C05441=1066.388,-25.189,-63.754,172.227,25.150,154.618
C05442=1066.394,-24.939,-63.767,172.229,25.153,154.619
C05443=1066.400,-24.690,-63.780,172.230,25.155,154.619
C05444=1066.407,-24.440,-63.794,172.232,25.157,154.619
C05445=1066.413,-24.190,-63.807,172.233,25.159,154.619
C05446=1066.418,-23.941,-63.821,172.235,25.162,154.620
C05447=1066.424,-23.691,-63.833,172.236,25.164,154.620
C05448=1066.431,-23.442,-63.847,172.238,25.166,154.620
C05449=1066.436,-23.192,-63.860,172.239,25.169,154.620
C05450=1066.442,-22.943,-63.874,172.240,25.171,154.621
C05451=1066.448,-22.694,-63.887,172.242,25.173,154.621
C05452=1066.454,-22.443,-63.901,172.243,25.176,154.621
C05453=1066.460,-22.193,-63.914,172.245,25.178,154.622
C05454=1066.467,-21.944,-63.927,172.246,25.181,154.622
C05455=1066.472,-21.695,-63.941,172.248,25.183,154.622
C05456=1066.478,-21.445,-63.954,172.249,25.185,154.622
C05457=1066.485,-21.196,-63.967,172.251,25.187,154.622
C05458=1066.491,-20.946,-63.982,172.252,25.189,154.623
C05459=1066.496,-20.696,-63.994,172.253,25.192,154.623
C05460=1066.503,-20.447,-64.008,172.255,25.194,154.623
C05461=1066.508,-20.197,-64.021,172.256,25.196,154.624
C05462=1066.514,-19.948,-64.035,172.258,25.199,154.624
C05463=1066.521,-19.698,-64.048,172.259,25.201,154.624
C05464=1066.527,-19.448,-64.062,172.261,25.204,154.624
C05465=1066.533,-19.199,-64.075,172.262,25.206,154.625
C05466=1066.539,-18.950,-64.089,172.263,25.208,154.625
C05467=1066.545,-18.700,-64.103,172.265,25.211,154.625
C05468=1066.551,-18.450,-64.116,172.266,25.213,154.625
C05469=1066.558,-18.172,-64.131,172.268,25.215,154.626
C05470=1066.564,-17.893,-64.146,172.270,25.218,154.626
C05471=1066.571,-17.615,-64.162,172.271,25.221,154.626
C05472=1066.578,-17.338,-64.176,172.273,25.223,154.627
C05473=1066.584,-17.087,-64.190,172.274,25.226,154.627
C05474=1066.591,-16.838,-64.204,172.276,25.228,154.627
C05475=1066.596,-16.589,-64.217,172.277,25.230,154.627
C05476=1066.602,-16.339,-64.231,172.279,25.233,154.628
C05477=1066.609,-16.089,-64.244,172.280,25.235,154.628
C05478=1066.615,-15.840,-64.258,172.282,25.237,154.628
C05479=1066.621,-15.590,-64.272,172.283,25.240,154.628
C05480=1066.627,-15.341,-64.285,172.284,25.242,154.629
C05481=1066.633,-15.091,-64.299,172.286,25.244,154.629
C05482=1066.639,-14.842,-64.312,172.287,25.247,154.629
C05483=1066.645,-14.592,-64.326,172.289,25.249,154.630
C05484=1066.651,-14.342,-64.340,172.290,25.252,154.630
C05485=1066.657,-14.093,-64.354,172.292,25.254,154.630
C05486=1066.663,-13.843,-64.368,172.294,25.257,154.630
C05487=1066.669,-13.594,-64.381,172.295,25.259,154.631
C05488=1066.675,-13.345,-64.395,172.297,25.261,154.631
C05489=1066.681,-13.095,-64.409,172.298,25.264,154.631
C05490=1066.687,-12.845,-64.423,172.300,25.267,154.632
C05491=1066.692,-12.596,-64.437,172.301,25.269,154.632
C05492=1066.699,-12.346,-64.450,172.302,25.271,154.632
C05493=1066.705,-12.096,-64.464,172.304,25.274,154.632
C05494=1066.711,-11.847,-64.478,172.305,25.276,154.633
C05495=1066.717,-11.598,-64.492,172.307,25.278,154.633
C05496=1066.723,-11.348,-64.506,172.308,25.281,154.633
C05497=1066.729,-11.098,-64.520,172.310,25.283,154.633
C05498=1066.734,-10.849,-64.533,172.311,25.286,154.634
C05499=1066.741,-10.599,-64.547,172.312,25.288,154.634
C05500=1066.747,-10.350,-64.562,172.314,25.291,154.634
C05501=1066.752,-10.100,-64.576,172.315,25.293,154.635
C05502=1066.759,-9.850,-64.589,172.317,25.295,154.635
C05503=1066.765,-9.601,-64.603,172.318,25.298,154.635
C05504=1066.771,-9.352,-64.617,172.320,25.300,154.635
C05505=1066.777,-9.102,-64.631,172.321,25.302,154.636
C05506=1066.783,-8.852,-64.645,172.322,25.305,154.636
C05507=1066.789,-8.603,-64.658,172.324,25.308,154.636
C05508=1066.795,-8.353,-64.673,172.325,25.310,154.637
C05509=1066.801,-8.104,-64.687,172.327,25.312,154.637
C05510=1066.807,-7.854,-64.700,172.328,25.315,154.637
C05511=1066.813,-7.604,-64.715,172.330,25.317,154.637
C05512=1066.819,-7.355,-64.729,172.331,25.319,154.638
C05513=1066.825,-7.106,-64.743,172.332,25.322,154.638
C05514=1066.831,-6.856,-64.757,172.334,25.325,154.638
C05515=1066.837,-6.607,-64.771,172.335,25.327,154.639
C05516=1066.844,-6.357,-64.785,172.337,25.329,154.639
C05517=1066.849,-6.107,-64.799,172.338,25.332,154.639
C05518=1066.855,-5.858,-64.813,172.340,25.334,154.640
C05519=1066.862,-5.608,-64.827,172.341,25.336,154.640
C05520=1066.867,-5.359,-64.841,172.342,25.339,154.640
C05521=1066.875,-5.109,-64.855,172.344,25.342,154.640
C05522=1066.880,-4.860,-64.869,172.345,25.344,154.641
C05523=1066.886,-4.611,-64.884,172.347,25.346,154.641
C05524=1066.892,-4.361,-64.898,172.348,25.349,154.641
C05525=1066.898,-4.111,-64.911,172.349,25.351,154.642
C05526=1066.904,-3.862,-64.926,172.351,25.353,154.642
C05527=1066.910,-3.612,-64.940,172.352,25.356,154.642
C05528=1066.917,-3.363,-64.954,172.354,25.359,154.642
C05529=1066.923,-3.113,-64.968,172.355,25.361,154.643
C05530=1066.928,-2.864,-64.982,172.357,25.363,154.643
C05531=1066.934,-2.614,-64.997,172.358,25.366,154.643
C05532=1066.940,-2.364,-65.011,172.359,25.369,154.644
C05533=1066.947,-2.085,-65.027,172.361,25.371,154.644
C05534=1066.953,-1.805,-65.043,172.363,25.374,154.644
C05535=1066.960,-1.525,-65.059,172.364,25.377,154.645
C05536=1066.966,-1.245,-65.075,172.366,25.380,154.645
C05537=1066.973,-0.995,-65.089,172.367,25.382,154.645
C05538=1066.978,-0.746,-65.104,172.369,25.385,154.646
C05539=1066.984,-0.496,-65.118,172.370,25.388,154.646
C05540=1066.990,-0.247,-65.133,172.371,25.390,154.646
C05541=1066.996,0.003,-65.147,172.373,25.392,154.647
C05542=1067.002,0.252,-65.162,172.374,25.395,154.647
C05543=1067.008,0.501,-65.176,172.376,25.398,154.647
C05544=1067.014,0.752,-65.191,172.377,25.400,154.648
C05545=1067.020,1.001,-65.205,172.378,25.402,154.648
C05546=1067.025,1.250,-65.219,172.380,25.405,154.648
C05547=1067.032,1.500,-65.233,172.381,25.408,154.648
C05548=1067.038,1.749,-65.247,172.383,25.410,154.649
C05549=1067.044,1.999,-65.262,172.384,25.413,154.649
C05550=1067.050,2.248,-65.277,172.385,25.415,154.649
C05551=1067.056,2.498,-65.291,172.387,25.417,154.650
C05552=1067.062,2.747,-65.305,172.388,25.420,154.650
C05553=1067.068,2.997,-65.320,172.390,25.423,154.650
C05554=1067.074,3.246,-65.334,172.391,25.425,154.651
C05555=1067.080,3.496,-65.349,172.392,25.428,154.651
C05556=1067.085,3.745,-65.363,172.394,25.430,154.651
C05557=1067.092,3.995,-65.378,172.395,25.433,154.652
C05558=1067.098,4.244,-65.393,172.397,25.436,154.652
C05559=1067.104,4.494,-65.407,172.398,25.438,154.652
C05560=1067.109,4.743,-65.421,172.399,25.440,154.652
C05561=1067.116,4.993,-65.436,172.401,25.443,154.653
C05562=1067.121,5.243,-65.450,172.402,25.446,154.653
C05563=1067.128,5.492,-65.465,172.404,25.448,154.653
C05564=1067.134,5.741,-65.480,172.405,25.451,154.654
C05565=1067.140,5.991,-65.495,172.406,25.453,154.654
C05566=1067.145,6.240,-65.509,172.408,25.455,154.654
C05567=1067.152,6.490,-65.524,172.409,25.458,154.655
C05568=1067.158,6.739,-65.538,172.411,25.461,154.655
C05569=1067.164,6.989,-65.553,172.412,25.463,154.655
C05570=1067.169,7.238,-65.567,172.413,25.466,154.656
C05571=1067.176,7.488,-65.582,172.415,25.468,154.656
C05572=1067.181,7.738,-65.597,172.416,25.471,154.656
C05573=1067.187,7.987,-65.612,172.418,25.474,154.657
C05574=1067.193,8.237,-65.626,172.419,25.476,154.657
C05575=1067.199,8.486,-65.641,172.421,25.478,154.657
C05576=1067.205,8.736,-65.656,172.422,25.481,154.658
C05577=1067.215,9.138,-65.680,172.424,25.485,154.658
C05578=1067.225,9.540,-65.702,172.426,25.489,154.659
C05579=1067.235,9.942,-65.727,172.429,25.493,154.659
C05580=1067.245,10.344,-65.750,172.431,25.497,154.660
C05581=1067.251,10.594,-65.765,172.433,25.499,154.660
C05582=1067.257,10.843,-65.779,172.434,25.502,154.660
C05583=1067.263,11.093,-65.794,172.435,25.505,154.660
C05584=1067.269,11.343,-65.810,172.437,25.507,154.661
C05585=1067.275,11.592,-65.825,172.438,25.510,154.661
C05586=1067.281,11.841,-65.839,172.440,25.512,154.661
C05587=1067.287,12.090,-65.854,172.441,25.515,154.662
C05588=1067.293,12.340,-65.868,172.442,25.518,154.662
C05589=1067.299,12.590,-65.883,172.444,25.520,154.662
C05590=1067.305,12.839,-65.898,172.445,25.522,154.663
C05591=1067.311,13.089,-65.913,172.447,25.525,154.663
C05592=1067.318,13.338,-65.928,172.448,25.527,154.663
C05593=1067.327,13.716,-65.951,172.450,25.531,154.664
C05594=1067.336,14.095,-65.973,172.452,25.535,154.664
C05595=1067.345,14.475,-65.996,172.455,25.539,154.665
C05596=1067.354,14.853,-66.018,172.456,25.543,154.665
C05597=1067.361,15.102,-66.033,172.458,25.546,154.666
C05598=1067.366,15.352,-66.049,172.459,25.548,154.666
C05599=1067.372,15.601,-66.064,172.461,25.551,154.666
C05600=1067.378,15.850,-66.078,172.462,25.553,154.667
C05601=1067.384,16.100,-66.093,172.464,25.556,154.667
C05602=1067.390,16.350,-66.109,172.465,25.558,154.667
C05603=1067.396,16.599,-66.123,172.466,25.561,154.668
C05604=1067.402,16.848,-66.138,172.468,25.564,154.668
C05605=1067.408,17.098,-66.154,172.469,25.566,154.668
C05606=1067.414,17.347,-66.168,172.471,25.569,154.669
C05607=1067.420,17.597,-66.183,172.472,25.572,154.669
C05608=1067.426,17.847,-66.199,172.473,25.574,154.669
C05609=1067.431,18.096,-66.213,172.475,25.577,154.670
C05610=1067.438,18.345,-66.229,172.476,25.579,154.670
C05611=1067.444,18.595,-66.244,172.478,25.582,154.670
C05612=1067.450,18.845,-66.259,172.479,25.584,154.671
C05613=1067.456,19.094,-66.274,172.480,25.587,154.671
C05614=1067.462,19.344,-66.290,172.482,25.590,154.671
C05615=1067.468,19.593,-66.304,172.483,25.592,154.671
C05616=1067.474,19.842,-66.319,172.485,25.595,154.672
C05617=1067.480,20.092,-66.335,172.486,25.597,154.672
C05618=1067.486,20.341,-66.350,172.487,25.600,154.673
C05619=1067.492,20.591,-66.365,172.489,25.602,154.673
C05620=1067.498,20.840,-66.380,172.490,25.605,154.673
C05621=1067.504,21.090,-66.395,172.492,25.608,154.674
C05622=1067.510,21.340,-66.411,172.493,25.611,154.674
C05623=1067.516,21.588,-66.426,172.494,25.613,154.674
C05624=1067.521,21.838,-66.442,172.496,25.616,154.675
C05625=1067.528,22.088,-66.457,172.497,25.618,154.675
C05626=1067.533,22.338,-66.472,172.499,25.621,154.675
C05627=1067.539,22.586,-66.488,172.500,25.623,154.676
C05628=1067.546,22.836,-66.502,172.501,25.626,154.676
C05629=1067.551,23.086,-66.518,172.503,25.629,154.676
C05630=1067.557,23.335,-66.533,172.504,25.631,154.677
C05631=1067.563,23.584,-66.549,172.506,25.634,154.677
C05632=1067.570,23.834,-66.564,172.507,25.637,154.677
C05633=1067.575,24.084,-66.579,172.508,25.639,154.678
C05634=1067.581,24.332,-66.594,172.510,25.642,154.678
C05635=1067.587,24.582,-66.610,172.511,25.644,154.678
C05636=1067.593,24.831,-66.625,172.513,25.647,154.679
C05637=1067.599,25.081,-66.641,172.514,25.649,154.679
C05638=1067.606,25.331,-66.656,172.515,25.652,154.679
C05639=1067.611,25.580,-66.671,172.517,25.655,154.680
C05640=1067.617,25.829,-66.686,172.518,25.658,154.680
C05641=1067.623,26.079,-66.703,172.520,25.660,154.680
C05642=1067.629,26.328,-66.718,172.521,25.663,154.681
C05643=1067.635,26.578,-66.733,172.522,25.665,154.681
C05644=1067.641,26.827,-66.748,172.524,25.668,154.681
C05645=1067.647,27.077,-66.764,172.525,25.670,154.682
C05646=1067.653,27.326,-66.780,172.527,25.673,154.682
C05647=1067.659,27.576,-66.795,172.528,25.676,154.682
C05648=1067.665,27.825,-66.810,172.529,25.678,154.683
C05649=1067.671,28.074,-66.826,172.531,25.681,154.683
C05650=1067.676,28.324,-66.842,172.532,25.684,154.683
C05651=1067.683,28.573,-66.857,172.533,25.687,154.684
C05652=1067.689,28.823,-66.873,172.535,25.689,154.684
C05653=1067.695,29.072,-66.888,172.536,25.692,154.684
C05654=1067.701,29.322,-66.904,172.538,25.694,154.685
C05655=1067.706,29.571,-66.920,172.539,25.697,154.685
C05656=1067.713,29.820,-66.935,172.540,25.700,154.685
C05657=1067.720,30.103,-66.952,172.542,25.703,154.686
C05658=1067.726,30.387,-66.970,172.543,25.706,154.686
C05659=1067.733,30.670,-66.988,172.544,25.709,154.687
C05660=1067.740,30.954,-67.006,172.547,25.712,154.687
C05661=1067.745,31.202,-67.022,172.548,25.714,154.687
C05662=1067.751,31.452,-67.037,172.550,25.717,154.688
C05663=1067.757,31.702,-67.054,172.551,25.720,154.688
C05664=1067.763,31.951,-67.068,172.552,25.722,154.688
C05665=1067.769,32.201,-67.085,172.554,25.725,154.689
C05666=1067.775,32.451,-67.100,172.554,25.727,154.689
C05667=1067.782,32.700,-67.116,172.556,25.730,154.689
C05668=1067.787,32.948,-67.132,172.557,25.733,154.690
C05669=1067.793,33.198,-67.147,172.558,25.735,154.690
C05670=1067.799,33.448,-67.164,172.560,25.738,154.691
C05671=1067.805,33.697,-67.179,172.561,25.740,154.691
C05672=1067.811,33.947,-67.195,172.563,25.743,154.691
C05673=1067.817,34.196,-67.211,172.564,25.746,154.692
C05674=1067.823,34.446,-67.226,172.565,25.748,154.692
C05675=1067.829,34.695,-67.242,172.567,25.751,154.692
C05676=1067.835,34.945,-67.258,172.568,25.754,154.693
C05677=1067.840,35.194,-67.274,172.570,25.757,154.693
C05678=1067.847,35.443,-67.289,172.571,25.759,154.693
C05679=1067.853,35.693,-67.305,172.572,25.762,154.694
C05680=1067.859,35.942,-67.321,172.574,25.765,154.694
C05681=1067.864,36.191,-67.337,172.575,25.767,154.694
C05682=1067.871,36.441,-67.352,172.577,25.770,154.695
C05683=1067.877,36.690,-67.369,172.578,25.772,154.695
C05684=1067.883,36.940,-67.385,172.579,25.775,154.695
C05685=1067.888,37.190,-67.400,172.581,25.777,154.696
C05686=1067.895,37.439,-67.416,172.582,25.780,154.696
C05687=1067.901,37.688,-67.432,172.584,25.783,154.696
C05688=1067.907,37.937,-67.449,172.585,25.785,154.697
C05689=1067.913,38.187,-67.464,172.586,25.788,154.697
C05690=1067.919,38.437,-67.480,172.588,25.791,154.697
C05691=1067.924,38.685,-67.496,172.589,25.794,154.698
C05692=1067.930,38.935,-67.513,172.591,25.796,154.698
C05693=1067.936,39.185,-67.528,172.592,25.799,154.698
C05694=1067.941,39.434,-67.544,172.593,25.802,154.699
C05695=1067.947,39.683,-67.561,172.595,25.805,154.699
C05696=1067.953,39.933,-67.577,172.596,25.807,154.700
C05697=1067.960,40.182,-67.593,172.598,25.810,154.700
C05698=1067.966,40.432,-67.608,172.599,25.813,154.700
C05699=1067.972,40.681,-67.624,172.600,25.815,154.701
C05700=1067.978,40.930,-67.641,172.602,25.818,154.701
C05701=1067.984,41.180,-67.657,172.603,25.821,154.701
C05702=1067.990,41.429,-67.673,172.605,25.823,154.702
C05703=1067.995,41.678,-67.689,172.606,25.826,154.702
C05704=1068.001,41.928,-67.705,172.607,25.829,154.702
C05705=1068.007,42.178,-67.721,172.609,25.831,154.703
C05706=1068.013,42.427,-67.737,172.610,25.834,154.703
C05707=1068.019,42.676,-67.754,172.611,25.837,154.704
C05708=1068.025,42.926,-67.770,172.613,25.839,154.704
C05709=1068.031,43.175,-67.786,172.614,25.842,154.704
C05710=1068.037,43.424,-67.802,172.616,25.844,154.705
C05711=1068.043,43.674,-67.819,172.617,25.847,154.705
C05712=1068.049,43.923,-67.835,172.618,25.850,154.705
C05713=1068.054,44.173,-67.850,172.620,25.853,154.706
C05714=1068.060,44.422,-67.867,172.621,25.855,154.706
C05715=1068.066,44.672,-67.884,172.623,25.858,154.706
C05716=1068.071,44.921,-67.900,172.624,25.861,154.707
C05717=1068.077,45.170,-67.916,172.625,25.864,154.707
C05718=1068.083,45.419,-67.932,172.627,25.866,154.707
C05719=1068.089,45.669,-67.948,172.628,25.869,154.708
C05720=1068.095,45.918,-67.964,172.630,25.872,154.708
C05721=1068.101,46.202,-67.984,172.631,25.875,154.709
C05722=1068.107,46.485,-68.002,172.633,25.878,154.709
C05723=1068.114,46.768,-68.020,172.634,25.881,154.710
C05724=1068.121,47.051,-68.040,172.636,25.884,154.710
C05725=1068.127,47.301,-68.056,172.637,25.887,154.710
C05726=1068.133,47.550,-68.072,172.639,25.890,154.711
C05727=1068.139,47.799,-68.089,172.640,25.892,154.711
C05728=1068.144,48.049,-68.105,172.641,25.895,154.711
C05729=1068.150,48.298,-68.122,172.643,25.898,154.712
C05730=1068.156,48.548,-68.138,172.644,25.900,154.712
C05731=1068.162,48.797,-68.154,172.646,25.903,154.712
C05732=1068.167,49.047,-68.171,172.647,25.906,154.713
C05733=1068.173,49.296,-68.187,172.648,25.909,154.713
C05734=1068.179,49.545,-68.204,172.650,25.911,154.714
C05735=1068.185,49.794,-68.221,172.651,25.914,154.714
C05736=1068.191,50.043,-68.237,172.653,25.917,154.714
C05737=1068.197,50.293,-68.254,172.654,25.919,154.715
C05738=1068.203,50.543,-68.270,172.655,25.922,154.715
C05739=1068.209,50.792,-68.286,172.657,25.925,154.715
C05740=1068.215,51.042,-68.303,172.658,25.927,154.716
C05741=1068.220,51.292,-68.320,172.660,25.930,154.716
C05742=1068.227,51.540,-68.337,172.661,25.933,154.716
C05743=1068.233,51.790,-68.353,172.662,25.936,154.717
C05744=1068.238,52.039,-68.369,172.664,25.938,154.717
C05745=1068.244,52.289,-68.386,172.665,25.941,154.718
C05746=1068.250,52.538,-68.402,172.667,25.944,154.718
C05747=1068.256,52.787,-68.418,172.668,25.946,154.718
C05748=1068.262,53.036,-68.435,172.669,25.949,154.719
C05749=1068.267,53.286,-68.452,172.671,25.952,154.719
C05750=1068.274,53.536,-68.469,172.672,25.955,154.719
C05751=1068.280,53.785,-68.485,172.674,25.957,154.720
C05752=1068.286,54.034,-68.502,172.675,25.960,154.720
C05753=1068.291,54.284,-68.519,172.676,25.963,154.720
C05754=1068.297,54.533,-68.535,172.678,25.965,154.721
C05755=1068.303,54.782,-68.552,172.679,25.968,154.721
C05756=1068.308,55.031,-68.569,172.681,25.971,154.722
C05757=1068.315,55.281,-68.586,172.682,25.973,154.722
C05758=1068.321,55.531,-68.602,172.683,25.976,154.722
C05759=1068.327,55.779,-68.619,172.685,25.979,154.723
C05760=1068.332,56.029,-68.636,172.686,25.982,154.723
C05761=1068.338,56.278,-68.652,172.688,25.984,154.723
C05762=1068.345,56.527,-68.669,172.689,25.987,154.724
C05763=1068.350,56.777,-68.686,172.690,25.990,154.724
C05764=1068.356,57.027,-68.702,172.692,25.992,154.724
C05765=1068.363,57.276,-68.719,172.693,25.995,154.725
C05766=1068.369,57.525,-68.736,172.695,25.998,154.725
C05767=1068.374,57.775,-68.753,172.696,26.000,154.726
C05768=1068.381,58.024,-68.770,172.697,26.003,154.726
C05769=1068.387,58.273,-68.786,172.699,26.006,154.726
C05770=1068.392,58.523,-68.803,172.700,26.008,154.727
C05771=1068.398,58.772,-68.820,172.703,26.011,154.727
C05772=1068.405,59.022,-68.837,172.704,26.014,154.727
C05773=1068.410,59.271,-68.854,172.705,26.017,154.728
C05774=1068.416,59.520,-68.870,172.707,26.019,154.728
C05775=1068.422,59.770,-68.887,172.708,26.022,154.728
C05776=1068.428,60.019,-68.905,172.710,26.025,154.729
C05777=1068.434,60.269,-68.921,172.711,26.027,154.729
C05778=1068.440,60.517,-68.938,172.713,26.030,154.729
C05779=1068.446,60.767,-68.955,172.714,26.033,154.730
C05780=1068.452,61.016,-68.972,172.715,26.035,154.730
C05781=1068.458,61.266,-68.988,172.717,26.038,154.730
C05782=1068.464,61.515,-69.006,172.718,26.041,154.731
C05783=1068.470,61.764,-69.022,172.720,26.043,154.731
C05784=1068.477,62.014,-69.039,172.721,26.046,154.732
C05785=1068.483,62.296,-69.058,172.722,26.049,154.732
C05786=1068.490,62.580,-69.078,172.724,26.052,154.732
C05787=1068.496,62.862,-69.097,172.726,26.055,154.733
C05788=1068.504,63.145,-69.116,172.727,26.058,154.733
C05789=1068.509,63.395,-69.134,172.729,26.061,154.734
C05790=1068.516,63.645,-69.150,172.730,26.063,154.734
C05791=1068.521,63.894,-69.168,172.732,26.066,154.734
C05792=1068.527,64.143,-69.184,172.733,26.069,154.735
C05793=1068.534,64.392,-69.202,172.735,26.071,154.735
C05794=1068.539,64.642,-69.218,172.736,26.074,154.735
C05795=1068.546,64.891,-69.235,172.737,26.077,154.736
C05796=1068.551,65.140,-69.253,172.739,26.079,154.736
C05797=1068.557,65.390,-69.270,172.740,26.082,154.736
C05798=1068.563,65.639,-69.287,172.742,26.085,154.737
C05799=1068.568,65.889,-69.304,172.743,26.088,154.737
C05800=1068.575,66.138,-69.321,172.744,26.090,154.737
C05801=1068.581,66.387,-69.339,172.746,26.093,154.738
C05802=1068.586,66.637,-69.356,172.747,26.096,154.738
C05803=1068.592,66.885,-69.373,172.749,26.098,154.739
C05804=1068.598,67.135,-69.391,172.750,26.101,154.739
C05805=1068.604,67.385,-69.407,172.751,26.104,154.739
C05806=1068.610,67.634,-69.424,172.753,26.107,154.740
C05807=1068.616,67.883,-69.442,172.754,26.109,154.740
C05808=1068.622,68.133,-69.459,172.756,26.112,154.740
C05809=1068.628,68.382,-69.476,172.757,26.115,154.741
C05810=1068.634,68.631,-69.494,172.759,26.117,154.741
C05811=1068.640,68.880,-69.511,172.760,26.120,154.741
C05812=1068.645,69.130,-69.528,172.761,26.123,154.742
C05813=1068.651,69.380,-69.546,172.763,26.125,154.742
C05814=1068.657,69.628,-69.563,172.764,26.128,154.743
C05815=1068.663,69.877,-69.580,172.767,26.131,154.743
C05816=1068.669,70.128,-69.598,172.768,26.134,154.743
C05817=1068.675,70.376,-69.615,172.769,26.137,154.744
C05818=1068.681,70.625,-69.632,172.771,26.139,154.744
C05819=1068.687,70.875,-69.650,172.772,26.142,154.744
C05820=1068.692,71.124,-69.668,172.774,26.145,154.745
C05821=1068.698,71.374,-69.684,172.775,26.147,154.745
C05822=1068.704,71.623,-69.702,172.776,26.150,154.745
C05823=1068.710,71.872,-69.719,172.778,26.153,154.746
C05824=1068.715,72.121,-69.737,172.779,26.155,154.746
C05825=1068.722,72.371,-69.754,172.781,26.158,154.747
C05826=1068.728,72.620,-69.772,172.782,26.161,154.747
C05827=1068.734,72.870,-69.789,172.783,26.163,154.747
C05828=1068.739,73.119,-69.807,172.785,26.166,154.748
C05829=1068.745,73.368,-69.824,172.786,26.169,154.748
C05830=1068.751,73.618,-69.842,172.788,26.171,154.748
C05831=1068.757,73.867,-69.859,172.789,26.174,154.749
C05832=1068.762,74.116,-69.877,172.791,26.177,154.749
C05833=1068.769,74.366,-69.895,172.792,26.179,154.750
C05834=1068.774,74.615,-69.912,172.793,26.182,154.750
C05835=1068.780,74.864,-69.930,172.795,26.185,154.750
C05836=1068.786,75.113,-69.947,172.796,26.188,154.751
C05837=1068.792,75.362,-69.965,172.798,26.190,154.751
C05838=1068.798,75.612,-69.983,172.799,26.193,154.751
C05839=1068.803,75.862,-70.000,172.800,26.196,154.752
C05840=1068.809,76.111,-70.017,172.802,26.198,154.752
C05841=1068.815,76.360,-70.035,172.803,26.201,154.753
C05842=1068.822,76.610,-70.052,172.805,26.204,154.753
C05843=1068.827,76.859,-70.070,172.806,26.207,154.753
C05844=1068.833,77.109,-70.088,172.808,26.209,154.754
C05845=1068.839,77.358,-70.105,172.810,26.212,154.754
C05846=1068.845,77.607,-70.123,172.811,26.215,154.754
C05847=1068.851,77.856,-70.141,172.813,26.217,154.755
C05848=1068.856,78.105,-70.158,172.814,26.220,154.755
C05849=1068.863,78.388,-70.179,172.816,26.223,154.755
C05850=1068.870,78.671,-70.199,172.817,26.227,154.756
C05851=1068.876,78.954,-70.219,172.819,26.230,154.756
C05852=1068.883,79.237,-70.239,172.821,26.233,154.757
C05853=1068.889,79.486,-70.256,172.822,26.235,154.757
C05854=1068.895,79.735,-70.275,172.823,26.238,154.758
C05855=1068.901,79.984,-70.293,172.825,26.241,154.758
C05856=1068.907,80.234,-70.311,172.826,26.243,154.758
C05857=1068.912,80.483,-70.328,172.828,26.246,154.759
C05858=1068.919,80.732,-70.346,172.829,26.249,154.759
C05859=1068.923,80.982,-70.364,172.830,26.252,154.759
C05860=1068.929,81.232,-70.382,172.832,26.255,154.760
C05861=1068.935,81.481,-70.400,172.833,26.257,154.760
C05862=1068.941,81.729,-70.418,172.835,26.260,154.761
C05863=1068.947,81.979,-70.436,172.836,26.263,154.761
C05864=1068.952,82.228,-70.454,172.838,26.266,154.761
C05865=1068.959,82.478,-70.472,172.840,26.268,154.762
C05866=1068.964,82.727,-70.489,172.841,26.271,154.762
C05867=1068.970,82.976,-70.508,172.843,26.274,154.762
C05868=1068.976,83.225,-70.525,172.844,26.277,154.763
C05869=1068.982,83.474,-70.543,172.846,26.279,154.763
C05870=1068.988,83.724,-70.561,172.847,26.282,154.763
C05871=1068.993,83.974,-70.579,172.848,26.285,154.764
C05872=1068.999,84.222,-70.598,172.850,26.288,154.764
C05873=1069.005,84.472,-70.616,172.851,26.290,154.765
C05874=1069.010,84.721,-70.633,172.853,26.293,154.765
C05875=1069.017,84.971,-70.651,172.854,26.295,154.765
C05876=1069.023,85.220,-70.670,172.856,26.298,154.766
C05877=1069.029,85.469,-70.687,172.857,26.301,154.766
C05878=1069.035,85.718,-70.705,172.858,26.303,154.766
C05879=1069.040,85.967,-70.723,172.860,26.306,154.767
C05880=1069.046,86.217,-70.742,172.861,26.309,154.767
C05881=1069.051,86.466,-70.760,172.863,26.311,154.768
C05882=1069.058,86.715,-70.778,172.865,26.315,154.768
C05883=1069.063,86.964,-70.796,172.866,26.317,154.768
C05884=1069.069,87.214,-70.814,172.868,26.320,154.769
C05885=1069.076,87.463,-70.832,172.869,26.323,154.769
C05886=1069.081,87.712,-70.850,172.871,26.325,154.769
C05887=1069.088,87.962,-70.868,172.872,26.328,154.770
C05888=1069.093,88.210,-70.887,172.874,26.331,154.770
C05889=1069.099,88.460,-70.905,172.875,26.333,154.770
C05890=1069.105,88.710,-70.923,172.876,26.336,154.771
C05891=1069.111,88.958,-70.941,172.878,26.338,154.771
C05892=1069.117,89.208,-70.959,172.879,26.341,154.772
C05893=1069.123,89.457,-70.977,172.881,26.344,154.772
C05894=1069.129,89.706,-70.995,172.882,26.346,154.772
C05895=1069.134,89.956,-71.014,172.884,26.349,154.773
C05896=1069.140,90.205,-71.032,172.886,26.352,154.773
C05897=1069.146,90.454,-71.050,172.888,26.355,154.773
C05898=1069.152,90.704,-71.068,172.889,26.358,154.774
C05899=1069.158,90.953,-71.086,172.890,26.360,154.774
C05900=1069.164,91.202,-71.105,172.892,26.363,154.774
C05901=1069.169,91.451,-71.123,172.893,26.365,154.775
C05902=1069.175,91.701,-71.142,172.895,26.368,154.775
C05903=1069.181,91.950,-71.160,172.896,26.371,154.776
C05904=1069.187,92.199,-71.178,172.898,26.374,154.776
C05905=1069.192,92.449,-71.197,172.899,26.377,154.776
C05906=1069.198,92.697,-71.215,172.900,26.379,154.777
C05907=1069.204,92.947,-71.233,172.902,26.382,154.777
C05908=1069.210,93.196,-71.252,172.903,26.385,154.777
C05909=1069.215,93.445,-71.270,172.905,26.388,154.778
C05910=1069.221,93.695,-71.289,172.907,26.390,154.778
C05911=1069.227,93.943,-71.307,172.908,26.393,154.779
C05912=1069.233,94.193,-71.325,172.910,26.396,154.779
C05913=1069.240,94.476,-71.347,172.911,26.399,154.779
C05914=1069.246,94.759,-71.367,172.913,26.402,154.780
C05915=1069.253,95.041,-71.389,172.915,26.405,154.780
C05916=1069.259,95.325,-71.409,172.916,26.408,154.781
C05917=1069.266,95.574,-71.428,172.918,26.411,154.781
C05918=1069.271,95.823,-71.447,172.919,26.413,154.781
C05919=1069.277,96.072,-71.465,172.921,26.416,154.782
C05920=1069.282,96.322,-71.484,172.923,26.419,154.782
C05921=1069.288,96.570,-71.502,172.924,26.422,154.782
C05922=1069.294,96.820,-71.521,172.926,26.424,154.783
C05923=1069.300,97.069,-71.539,172.927,26.427,154.783
C05924=1069.306,97.318,-71.558,172.929,26.430,154.784
C05925=1069.311,97.568,-71.576,172.930,26.433,154.784
C05926=1069.318,97.817,-71.595,172.932,26.435,154.784
C05927=1069.323,98.066,-71.614,172.933,26.438,154.785
C05928=1069.329,98.315,-71.632,172.935,26.441,154.785
C05929=1069.335,98.565,-71.651,172.936,26.443,154.785
C05930=1069.341,98.814,-71.670,172.937,26.446,154.786
C05931=1069.346,99.063,-71.689,172.940,26.449,154.786
C05932=1069.352,99.312,-71.706,172.941,26.451,154.786
C05933=1069.359,99.562,-71.725,172.943,26.454,154.787
C05934=1069.364,99.811,-71.744,172.944,26.457,154.787
C05935=1069.370,100.059,-71.763,172.946,26.460,154.788
C05936=1069.376,100.309,-71.782,172.947,26.462,154.788
C05937=1069.382,100.559,-71.800,172.948,26.465,154.788
C05938=1069.388,100.808,-71.819,172.950,26.468,154.789
C05939=1069.394,101.057,-71.838,172.951,26.470,154.789
C05940=1069.399,101.306,-71.857,172.954,26.473,154.789
C05941=1069.405,101.555,-71.876,172.955,26.476,154.790
C05942=1069.411,101.805,-71.894,172.957,26.479,154.790
C05943=1069.416,102.054,-71.913,172.958,26.481,154.790
C05944=1069.422,102.303,-71.932,172.960,26.484,154.791
C05945=1069.428,102.552,-71.951,172.961,26.487,154.791
C05946=1069.434,102.802,-71.970,172.962,26.489,154.792
C05947=1069.439,103.051,-71.989,172.964,26.492,154.792
C05948=1069.445,103.300,-72.007,172.965,26.495,154.792
C05949=1069.451,103.549,-72.027,172.967,26.497,154.793
C05950=1069.457,103.799,-72.046,172.969,26.500,154.793
C05951=1069.462,104.048,-72.063,172.970,26.503,154.794
C05952=1069.468,104.297,-72.083,172.972,26.506,154.794
C05953=1069.474,104.546,-72.102,172.973,26.508,154.794
C05954=1069.480,104.796,-72.120,172.975,26.511,154.795
C05955=1069.486,105.045,-72.140,172.976,26.514,154.795
C05956=1069.491,105.294,-72.159,172.978,26.516,154.795
C05957=1069.497,105.543,-72.177,172.979,26.519,154.796
C05958=1069.503,105.792,-72.196,172.982,26.522,154.796
C05959=1069.509,106.042,-72.216,172.983,26.525,154.797
C05960=1069.514,106.291,-72.235,172.984,26.527,154.797
C05961=1069.520,106.540,-72.253,172.986,26.530,154.797
C05962=1069.526,106.789,-72.272,172.987,26.533,154.798
C05963=1069.532,107.038,-72.292,172.989,26.535,154.798
C05964=1069.538,107.288,-72.310,172.990,26.538,154.798
C05965=1069.544,107.537,-72.330,172.992,26.541,154.799
C05966=1069.549,107.786,-72.348,172.994,26.544,154.799
C05967=1069.554,108.035,-72.368,172.996,26.546,154.799
C05968=1069.561,108.284,-72.386,172.997,26.549,154.800
C05969=1069.567,108.534,-72.406,172.998,26.552,154.800
C05970=1069.573,108.782,-72.426,173.000,26.554,154.800
C05971=1069.578,109.032,-72.445,173.001,26.557,154.801
C05972=1069.585,109.281,-72.463,173.003,26.560,154.801
C05973=1069.590,109.530,-72.483,173.004,26.562,154.802
C05974=1069.595,109.779,-72.502,173.007,26.565,154.802
C05975=1069.601,110.029,-72.521,173.008,26.568,154.802
C05976=1069.608,110.278,-72.539,173.009,26.571,154.803
C05977=1069.614,110.561,-72.561,173.011,26.574,154.803
C05978=1069.621,110.844,-72.583,173.013,26.577,154.803
C05979=1069.628,111.126,-72.605,173.015,26.580,154.804
C05980=1069.634,111.409,-72.627,173.017,26.583,154.804
C05981=1069.639,111.658,-72.646,173.018,26.586,154.805
C05982=1069.645,111.908,-72.666,173.020,26.588,154.805
C05983=1069.652,112.157,-72.684,173.021,26.591,154.805
C05984=1069.657,112.406,-72.704,173.023,26.594,154.806
C05985=1069.663,112.655,-72.724,173.024,26.596,154.806
C05986=1069.669,112.905,-72.743,173.026,26.599,154.807
C05987=1069.675,113.154,-72.762,173.028,26.602,154.807
C05988=1069.680,113.404,-72.781,173.030,26.605,154.807
C05989=1069.686,113.652,-72.801,173.031,26.607,154.808
C05990=1069.691,113.901,-72.820,173.033,26.610,154.808
C05991=1069.697,114.150,-72.839,173.034,26.612,154.808
C05992=1069.703,114.399,-72.859,173.035,26.615,154.809
C05993=1069.709,114.649,-72.879,173.038,26.618,154.809
C05994=1069.714,114.898,-72.898,173.039,26.621,154.810
C05995=1069.720,115.148,-72.917,173.041,26.623,154.810
C05996=1069.726,115.396,-72.937,173.042,26.626,154.810
C05997=1069.732,115.646,-72.956,173.044,26.629,154.811
C05998=1069.737,115.895,-72.976,173.045,26.632,154.811
C05999=1069.743,116.143,-72.995,173.046,26.635,154.811
C06000=1069.749,116.393,-73.014,173.049,26.637,154.812
C06001=1069.755,116.642,-73.034,173.050,26.640,154.812
C06002=1069.760,116.891,-73.054,173.052,26.643,154.812
C06003=1069.765,117.141,-73.073,173.053,26.646,154.813
C06004=1069.771,117.390,-73.093,173.055,26.649,154.813
C06005=1069.777,117.639,-73.113,173.056,26.651,154.814
C06006=1069.783,117.888,-73.133,173.059,26.654,154.814
C06007=1069.789,118.137,-73.152,173.060,26.657,154.814
C06008=1069.794,118.387,-73.171,173.061,26.660,154.815
C06009=1069.800,118.636,-73.191,173.063,26.662,154.815
C06010=1069.805,118.885,-73.211,173.064,26.665,154.815
C06011=1069.811,119.134,-73.231,173.066,26.667,154.816
C06012=1069.817,119.384,-73.250,173.068,26.671,154.816
C06013=1069.822,119.632,-73.270,173.070,26.673,154.817
C06014=1069.828,119.881,-73.289,173.071,26.676,154.817
C06015=1069.834,120.130,-73.309,173.073,26.678,154.817
C06016=1069.839,120.380,-73.329,173.074,26.681,154.818
C06017=1069.845,120.628,-73.349,173.075,26.684,154.818
C06018=1069.851,120.878,-73.368,173.078,26.687,154.818
C06019=1069.857,121.127,-73.388,173.079,26.689,154.819
C06020=1069.862,121.376,-73.407,173.081,26.692,154.819
C06021=1069.868,121.625,-73.427,173.082,26.695,154.820
C06022=1069.873,121.875,-73.447,173.084,26.697,154.820
C06023=1069.879,122.124,-73.467,173.086,26.700,154.820
C06024=1069.885,122.372,-73.487,173.088,26.703,154.821
C06025=1069.891,122.622,-73.506,173.089,26.705,154.821
C06026=1069.897,122.871,-73.526,173.090,26.708,154.821
C06027=1069.903,123.121,-73.546,173.092,26.711,154.822
C06028=1069.908,123.370,-73.566,173.094,26.714,154.822
C06029=1069.914,123.619,-73.586,173.096,26.716,154.822
C06030=1069.920,123.868,-73.605,173.097,26.719,154.823
C06031=1069.926,124.117,-73.625,173.099,26.722,154.823
C06032=1069.932,124.366,-73.645,173.100,26.724,154.824
C06033=1069.937,124.615,-73.665,173.103,26.727,154.824
C06034=1069.943,124.864,-73.685,173.104,26.730,154.824
C06035=1069.949,125.114,-73.704,173.105,26.733,154.825
C06036=1069.955,125.362,-73.724,173.107,26.735,154.825
C06037=1069.961,125.611,-73.744,173.108,26.738,154.825
C06038=1069.966,125.861,-73.764,173.111,26.741,154.826
C06039=1069.972,126.110,-73.784,173.112,26.743,154.826
C06040=1069.978,126.359,-73.804,173.114,26.746,154.826
C06041=1069.985,126.642,-73.827,173.115,26.749,154.827
C06042=1069.991,126.925,-73.849,173.118,26.752,154.827
C06043=1069.997,127.208,-73.872,173.119,26.755,154.828
C06044=1070.004,127.491,-73.895,173.121,26.759,154.828
C06045=1070.010,127.739,-73.915,173.123,26.761,154.828
C06046=1070.016,127.989,-73.934,173.124,26.764,154.829
C06047=1070.021,128.238,-73.955,173.127,26.767,154.829
C06048=1070.027,128.487,-73.975,173.128,26.769,154.829
C06049=1070.034,128.736,-73.995,173.130,26.772,154.830
C06050=1070.040,128.985,-74.015,173.131,26.774,154.830
C06051=1070.045,129.235,-74.035,173.134,26.777,154.831
C06052=1070.051,129.484,-74.055,173.135,26.780,154.831
C06053=1070.057,129.733,-74.075,173.137,26.782,154.831
C06054=1070.063,129.981,-74.095,173.138,26.785,154.832
C06055=1070.068,130.231,-74.116,173.139,26.788,154.832
C06056=1070.074,130.480,-74.136,173.142,26.790,154.832
C06057=1070.080,130.729,-74.155,173.143,26.793,154.833
C06058=1070.086,130.978,-74.175,173.145,26.795,154.833
C06059=1070.091,131.227,-74.195,173.146,26.798,154.833
C06060=1070.098,131.477,-74.216,173.149,26.801,154.834
C06061=1070.104,131.726,-74.236,173.150,26.804,154.834
C06062=1070.109,131.975,-74.256,173.152,26.806,154.834
C06063=1070.115,132.224,-74.276,173.153,26.809,154.835
C06064=1070.121,132.473,-74.297,173.156,26.812,154.835
C06065=1070.127,132.722,-74.317,173.157,26.815,154.836
C06066=1070.132,132.971,-74.338,173.159,26.817,154.836
C06067=1070.138,133.220,-74.358,173.160,26.820,154.836
C06068=1070.144,133.469,-74.378,173.163,26.823,154.837
C06069=1070.150,133.718,-74.398,173.164,26.825,154.837
C06070=1070.155,133.967,-74.419,173.165,26.828,154.837
C06071=1070.161,134.217,-74.439,173.167,26.831,154.838
C06072=1070.167,134.466,-74.460,173.168,26.833,154.838
C06073=1070.173,134.715,-74.480,173.171,26.836,154.838
C06074=1070.178,134.964,-74.500,173.172,26.839,154.839
C06075=1070.184,135.213,-74.520,173.174,26.841,154.839
C06076=1070.190,135.463,-74.541,173.175,26.844,154.840
C06077=1070.196,135.711,-74.561,173.178,26.847,154.840
C06078=1070.201,135.960,-74.581,173.179,26.850,154.840
C06079=1070.206,136.210,-74.602,173.181,26.852,154.841
C06080=1070.213,136.459,-74.622,173.183,26.855,154.841
C06081=1070.218,136.708,-74.643,173.184,26.858,154.841
C06082=1070.224,136.957,-74.663,173.186,26.860,154.842
C06083=1070.229,137.206,-74.683,173.187,26.863,154.842
C06084=1070.236,137.455,-74.704,173.190,26.866,154.843
C06085=1070.242,137.704,-74.725,173.191,26.869,154.843
C06086=1070.247,137.953,-74.746,173.193,26.871,154.843
C06087=1070.253,138.202,-74.766,173.194,26.874,154.844
C06088=1070.259,138.452,-74.786,173.197,26.877,154.844
C06089=1070.265,138.701,-74.806,173.198,26.880,154.844
C06090=1070.270,138.949,-74.828,173.200,26.882,154.845
C06091=1070.275,139.198,-74.848,173.201,26.885,154.845
C06092=1070.282,139.448,-74.869,173.204,26.888,154.845
C06093=1070.287,139.697,-74.889,173.205,26.890,154.846
C06094=1070.293,139.946,-74.910,173.207,26.893,154.846
C06095=1070.299,140.195,-74.931,173.209,26.896,154.846
C06096=1070.305,140.444,-74.951,173.210,26.899,154.847
C06097=1070.310,140.693,-74.972,173.212,26.901,154.847
C06098=1070.315,140.942,-74.992,173.213,26.904,154.848
C06099=1070.322,141.191,-75.013,173.216,26.907,154.848
C06100=1070.327,141.440,-75.034,173.217,26.909,154.848
C06101=1070.333,141.690,-75.054,173.219,26.912,154.849
C06102=1070.338,141.939,-75.075,173.221,26.915,154.849
C06103=1070.345,142.188,-75.096,173.223,26.918,154.849
C06104=1070.350,142.437,-75.117,173.224,26.920,154.850
C06105=1070.357,142.719,-75.141,173.227,26.923,154.850
C06106=1070.363,143.002,-75.164,173.228,26.926,154.851
C06107=1070.369,143.285,-75.187,173.230,26.930,154.851
C06108=1070.376,143.567,-75.211,173.233,26.933,154.851
C06109=1070.381,143.817,-75.232,173.234,26.936,154.852
C06110=1070.387,144.066,-75.253,173.236,26.938,154.852
C06111=1070.393,144.315,-75.274,173.237,26.941,154.853
C06112=1070.399,144.564,-75.294,173.240,26.944,154.853
C06113=1070.405,144.813,-75.315,173.241,26.946,154.853
C06114=1070.410,145.062,-75.336,173.243,26.949,154.854
C06115=1070.416,145.311,-75.358,173.245,26.952,154.854
C06116=1070.422,145.560,-75.378,173.247,26.954,154.854
C06117=1070.427,145.809,-75.399,173.248,26.957,154.855
C06118=1070.434,146.058,-75.420,173.250,26.960,154.855
C06119=1070.439,146.307,-75.441,173.252,26.963,154.855
C06120=1070.445,146.556,-75.462,173.253,26.965,154.856
C06121=1070.450,146.806,-75.482,173.256,26.968,154.856
C06122=1070.456,147.054,-75.504,173.257,26.971,154.857
C06123=1070.462,147.304,-75.525,173.259,26.973,154.857
C06124=1070.468,147.552,-75.545,173.261,26.976,154.857
C06125=1070.473,147.801,-75.566,173.263,26.979,154.858
C06126=1070.480,148.051,-75.588,173.264,26.981,154.858
C06127=1070.485,148.299,-75.609,173.266,26.984,154.858
C06128=1070.491,148.549,-75.630,173.268,26.987,154.859
C06129=1070.497,148.798,-75.651,173.270,26.990,154.859
C06130=1070.502,149.047,-75.672,173.271,26.992,154.859
C06131=1070.508,149.296,-75.693,173.273,26.995,154.860
C06132=1070.513,149.545,-75.714,173.275,26.998,154.860
C06133=1070.519,149.794,-75.735,173.277,27.000,154.860
C06134=1070.525,150.043,-75.757,173.279,27.003,154.861
C06135=1070.531,150.293,-75.778,173.280,27.006,154.861
C06136=1070.536,150.541,-75.799,173.282,27.009,154.862
C06137=1070.542,150.790,-75.819,173.284,27.011,154.862
C06138=1070.548,151.039,-75.841,173.286,27.014,154.862
C06139=1070.553,151.288,-75.862,173.288,27.017,154.863
C06140=1070.559,151.538,-75.883,173.290,27.020,154.863
C06141=1070.565,151.786,-75.904,173.291,27.022,154.863
C06142=1070.571,152.035,-75.926,173.294,27.025,154.864
C06143=1070.576,152.285,-75.947,173.295,27.028,154.864
C06144=1070.582,152.533,-75.968,173.297,27.031,154.865
C06145=1070.588,152.782,-75.990,173.299,27.033,154.865
C06146=1070.593,153.031,-76.011,173.301,27.036,154.865
C06147=1070.599,153.281,-76.032,173.302,27.039,154.866
C06148=1070.604,153.529,-76.054,173.304,27.042,154.866
C06149=1070.610,153.779,-76.075,173.306,27.044,154.866
C06150=1070.616,154.027,-76.097,173.307,27.047,154.867
C06151=1070.622,154.277,-76.117,173.310,27.050,154.867
C06152=1070.627,154.525,-76.139,173.311,27.052,154.867
C06153=1070.633,154.775,-76.160,173.313,27.055,154.868
C06154=1070.639,155.023,-76.182,173.315,27.058,154.868
C06155=1070.645,155.272,-76.203,173.317,27.060,154.868
C06156=1070.650,155.521,-76.224,173.319,27.064,154.869
C06157=1070.656,155.771,-76.246,173.321,27.066,154.869
C06158=1070.661,156.019,-76.267,173.322,27.069,154.870
C06159=1070.668,156.269,-76.289,173.325,27.072,154.870
C06160=1070.673,156.517,-76.310,173.326,27.074,154.870
C06161=1070.679,156.766,-76.332,173.328,27.077,154.871
C06162=1070.684,157.015,-76.354,173.330,27.080,154.871
C06163=1070.690,157.265,-76.375,173.332,27.082,154.871
C06164=1070.696,157.514,-76.396,173.334,27.086,154.872
C06165=1070.702,157.763,-76.418,173.335,27.088,154.872
C06166=1070.707,158.012,-76.440,173.337,27.091,154.873
C06167=1070.713,158.261,-76.461,173.339,27.094,154.873
C06168=1070.719,158.510,-76.483,173.341,27.096,154.873
C06169=1070.725,158.793,-76.507,173.343,27.099,154.874
C06170=1070.731,159.074,-76.532,173.346,27.103,154.874
C06171=1070.738,159.357,-76.556,173.347,27.106,154.875
C06172=1070.744,159.639,-76.580,173.350,27.109,154.875
C06173=1070.750,159.889,-76.602,173.351,27.112,154.875
C06174=1070.756,160.137,-76.623,173.353,27.114,154.876
C06175=1070.761,160.387,-76.646,173.355,27.117,154.876
C06176=1070.768,160.636,-76.667,173.357,27.120,154.876
C06177=1070.773,160.884,-76.688,173.359,27.123,154.877
C06178=1070.779,161.134,-76.710,173.360,27.125,154.877
C06179=1070.784,161.382,-76.732,173.363,27.128,154.877
C06180=1070.790,161.632,-76.754,173.364,27.131,154.878
C06181=1070.795,161.880,-76.775,173.367,27.134,154.878
C06182=1070.802,162.129,-76.798,173.368,27.137,154.879
C06183=1070.807,162.379,-76.820,173.371,27.140,154.879
C06184=1070.812,162.627,-76.842,173.372,27.143,154.879
C06185=1070.818,162.877,-76.864,173.374,27.145,154.880
C06186=1070.823,163.125,-76.885,173.376,27.148,154.880
C06187=1070.829,163.375,-76.907,173.378,27.151,154.881
C06188=1070.834,163.623,-76.929,173.380,27.154,154.881
C06189=1070.840,163.872,-76.951,173.381,27.156,154.881
C06190=1070.845,164.121,-76.973,173.383,27.159,154.882
C06191=1070.850,164.370,-76.995,173.385,27.162,154.882
C06192=1070.857,164.620,-77.017,173.387,27.165,154.883
C06193=1070.861,164.868,-77.039,173.389,27.168,154.883
C06194=1070.868,165.117,-77.061,173.391,27.170,154.883
C06195=1070.873,165.366,-77.083,173.393,27.173,154.884
C06196=1070.878,165.615,-77.105,173.395,27.176,154.884
C06197=1070.884,165.864,-77.127,173.396,27.179,154.884
C06198=1070.889,166.113,-77.150,173.399,27.182,154.885
C06199=1070.896,166.362,-77.171,173.400,27.185,154.885
C06200=1070.900,166.611,-77.193,173.402,27.188,154.886
C06201=1070.906,166.860,-77.215,173.404,27.190,154.886
C06202=1070.912,167.109,-77.238,173.406,27.193,154.886
C06203=1070.917,167.358,-77.259,173.408,27.196,154.887
C06204=1070.923,167.607,-77.282,173.410,27.199,154.887
C06205=1070.929,167.856,-77.304,173.412,27.202,154.887
C06206=1070.934,168.105,-77.326,173.413,27.204,154.888
C06207=1070.940,168.354,-77.348,173.416,27.207,154.888
C06208=1070.946,168.603,-77.370,173.417,27.210,154.889
C06209=1070.951,168.851,-77.392,173.420,27.213,154.889
C06210=1070.957,169.101,-77.414,173.421,27.215,154.889
C06211=1070.963,169.350,-77.437,173.424,27.219,154.890
C06212=1070.967,169.598,-77.459,173.425,27.221,154.890
C06213=1070.974,169.847,-77.481,173.428,27.224,154.891
C06214=1070.979,170.096,-77.503,173.429,27.227,154.891
C06215=1070.984,170.345,-77.525,173.432,27.230,154.891
C06216=1070.991,170.594,-77.548,173.433,27.232,154.892
C06217=1070.996,170.843,-77.570,173.435,27.235,154.892
C06218=1071.002,171.092,-77.593,173.437,27.238,154.892
C06219=1071.007,171.341,-77.614,173.439,27.241,154.893
C06220=1071.013,171.590,-77.637,173.441,27.243,154.893
C06221=1071.018,171.839,-77.659,173.443,27.246,154.893
C06222=1071.025,172.088,-77.682,173.445,27.249,154.894
C06223=1071.030,172.337,-77.703,173.446,27.252,154.894
C06224=1071.035,172.585,-77.726,173.449,27.255,154.895
C06225=1071.042,172.835,-77.748,173.450,27.257,154.895
C06226=1071.047,173.084,-77.771,173.453,27.260,154.895
C06227=1071.052,173.332,-77.793,173.454,27.263,154.896
C06228=1071.058,173.581,-77.816,173.457,27.266,154.896
C06229=1071.064,173.831,-77.837,173.458,27.269,154.897
C06230=1071.070,174.079,-77.860,173.461,27.271,154.897
C06231=1071.075,174.328,-77.883,173.462,27.274,154.897
C06232=1071.081,174.577,-77.905,173.465,27.277,154.898
C06233=1071.087,174.859,-77.930,173.467,27.280,154.898
C06234=1071.094,175.141,-77.955,173.469,27.284,154.898
C06235=1071.100,175.423,-77.982,173.472,27.287,154.899
C06236=1071.107,175.705,-78.007,173.473,27.290,154.899
C06237=1071.113,175.954,-78.030,173.476,27.293,154.900
C06238=1071.119,176.203,-78.051,173.477,27.295,154.900
C06239=1071.124,176.452,-78.074,173.480,27.298,154.900
C06240=1071.130,176.701,-78.097,173.481,27.301,154.901
C06241=1071.136,176.951,-78.119,173.484,27.304,154.901
C06242=1071.141,177.198,-78.141,173.485,27.306,154.902
C06243=1071.147,177.447,-78.164,173.488,27.309,154.902
C06244=1071.153,177.697,-78.187,173.490,27.312,154.902
C06245=1071.158,177.946,-78.210,173.492,27.315,154.903
C06246=1071.164,178.195,-78.232,173.494,27.318,154.903
C06247=1071.171,178.443,-78.255,173.495,27.321,154.903
C06248=1071.176,178.693,-78.277,173.498,27.323,154.904
C06249=1071.182,178.942,-78.300,173.499,27.326,154.904
C06250=1071.187,179.191,-78.323,173.502,27.329,154.904
C06251=1071.194,179.439,-78.345,173.503,27.332,154.905
C06252=1071.199,179.688,-78.367,173.506,27.335,154.905
C06253=1071.204,179.937,-78.390,173.507,27.337,154.905
C06254=1071.210,180.186,-78.413,173.510,27.340,154.906
C06255=1071.216,180.435,-78.436,173.512,27.343,154.906
C06256=1071.222,180.683,-78.458,173.514,27.346,154.907
C06257=1071.228,180.932,-78.481,173.516,27.348,154.907
C06258=1071.234,181.181,-78.504,173.518,27.351,154.907
C06259=1071.239,181.431,-78.526,173.520,27.354,154.908
C06260=1071.245,181.679,-78.549,173.522,27.357,154.908
C06261=1071.251,181.928,-78.572,173.524,27.359,154.908
C06262=1071.257,182.177,-78.595,173.527,27.362,154.909
C06263=1071.263,182.426,-78.618,173.528,27.365,154.909
C06264=1071.269,182.675,-78.641,173.531,27.368,154.910
C06265=1071.274,182.924,-78.664,173.532,27.370,154.910
C06266=1071.281,183.172,-78.686,173.535,27.373,154.910
C06267=1071.287,183.421,-78.709,173.536,27.376,154.911
C06268=1071.292,183.670,-78.732,173.539,27.379,154.911
C06269=1071.298,183.919,-78.755,173.541,27.381,154.911
C06270=1071.304,184.168,-78.778,173.543,27.384,154.912
C06271=1071.310,184.417,-78.801,173.545,27.387,154.912
C06272=1071.315,184.666,-78.824,173.547,27.389,154.912
C06273=1071.321,184.914,-78.847,173.549,27.392,154.913
C06274=1071.327,185.163,-78.869,173.552,27.396,154.913
C06275=1071.332,185.412,-78.892,173.553,27.398,154.914
C06276=1071.338,185.661,-78.915,173.555,27.401,154.914
C06277=1071.343,185.910,-78.939,173.557,27.404,154.914
C06278=1071.349,186.159,-78.962,173.559,27.407,154.915
C06279=1071.355,186.408,-78.985,173.561,27.410,154.915
C06280=1071.360,186.657,-79.008,173.563,27.413,154.916
C06281=1071.365,186.906,-79.031,173.566,27.416,154.916
C06282=1071.371,187.155,-79.055,173.567,27.419,154.916
C06283=1071.377,187.403,-79.078,173.570,27.422,154.917
C06284=1071.382,187.653,-79.101,173.571,27.424,154.917
C06285=1071.388,187.902,-79.124,173.574,27.427,154.918
C06286=1071.394,188.150,-79.147,173.576,27.430,154.918
C06287=1071.399,188.399,-79.170,173.578,27.433,154.918
C06288=1071.405,188.648,-79.195,173.580,27.436,154.919
C06289=1071.410,188.897,-79.217,173.583,27.439,154.919
C06290=1071.416,189.146,-79.240,173.584,27.442,154.920
C06291=1071.421,189.395,-79.264,173.586,27.445,154.920
C06292=1071.427,189.643,-79.288,173.588,27.448,154.920
C06293=1071.433,189.892,-79.311,173.590,27.451,154.921
C06294=1071.439,190.141,-79.334,173.593,27.454,154.921
C06295=1071.444,190.390,-79.357,173.594,27.457,154.921
C06296=1071.450,190.638,-79.381,173.597,27.460,154.922
C06297=1071.456,190.920,-79.407,173.599,27.463,154.922
C06298=1071.462,191.202,-79.433,173.602,27.466,154.923
C06299=1071.468,191.484,-79.460,173.604,27.470,154.923
C06300=1071.475,191.766,-79.486,173.606,27.473,154.924
C06301=1071.481,192.014,-79.510,173.609,27.476,154.924
C06302=1071.486,192.263,-79.533,173.610,27.479,154.924
C06303=1071.492,192.512,-79.556,173.613,27.482,154.925
C06304=1071.498,192.760,-79.580,173.614,27.484,154.925
C06305=1071.503,193.009,-79.604,173.617,27.487,154.926
C06306=1071.509,193.258,-79.627,173.619,27.490,154.926
C06307=1071.514,193.508,-79.651,173.621,27.493,154.926
C06308=1071.520,193.757,-79.674,173.623,27.496,154.927
C06309=1071.526,194.005,-79.698,173.626,27.499,154.927
C06310=1071.531,194.254,-79.721,173.627,27.502,154.928
C06311=1071.537,194.502,-79.745,173.630,27.505,154.928
C06312=1071.543,194.751,-79.768,173.632,27.508,154.928
C06313=1071.548,195.000,-79.792,173.633,27.511,154.929
C06314=1071.554,195.249,-79.815,173.636,27.514,154.929
C06315=1071.560,195.498,-79.839,173.638,27.517,154.930
C06316=1071.565,195.747,-79.863,173.640,27.519,154.930
C06317=1071.571,195.995,-79.886,173.642,27.522,154.930
C06318=1071.576,196.244,-79.910,173.645,27.525,154.931
C06319=1071.582,196.493,-79.934,173.647,27.528,154.931
C06320=1071.589,196.742,-79.957,173.649,27.531,154.932
C06321=1071.594,196.991,-79.981,173.651,27.534,154.932
C06322=1071.600,197.240,-80.004,173.654,27.537,154.932
C06323=1071.605,197.488,-80.028,173.655,27.540,154.933
C06324=1071.611,197.737,-80.052,173.658,27.543,154.933
C06325=1071.617,197.986,-80.076,173.660,27.546,154.934
C06326=1071.623,198.235,-80.100,173.662,27.549,154.934
C06327=1071.629,198.484,-80.122,173.664,27.552,154.934
C06328=1071.634,198.732,-80.147,173.667,27.555,154.935
C06329=1071.640,198.981,-80.171,173.669,27.558,154.935
C06330=1071.645,199.230,-80.194,173.670,27.560,154.935
C06331=1071.651,199.479,-80.218,173.673,27.563,154.936
C06332=1071.657,199.727,-80.242,173.675,27.566,154.936
C06333=1071.663,199.977,-80.266,173.677,27.569,154.937
C06334=1071.669,200.225,-80.289,173.679,27.572,154.937
C06335=1071.674,200.474,-80.313,173.682,27.575,154.937
C06336=1071.681,200.722,-80.337,173.684,27.578,154.938
C06337=1071.686,200.972,-80.361,173.686,27.581,154.938
C06338=1071.692,201.220,-80.385,173.688,27.584,154.939
C06339=1071.697,201.469,-80.409,173.691,27.587,154.939
C06340=1071.704,201.718,-80.433,173.693,27.590,154.939
C06341=1071.709,201.967,-80.456,173.695,27.593,154.940
C06342=1071.715,202.215,-80.480,173.697,27.596,154.940
C06343=1071.721,202.465,-80.505,173.700,27.599,154.941
C06344=1071.727,202.713,-80.528,173.701,27.601,154.941
C06345=1071.732,202.961,-80.553,173.704,27.604,154.941
C06346=1071.738,203.210,-80.577,173.706,27.607,154.942
C06347=1071.743,203.460,-80.601,173.708,27.610,154.942
C06348=1071.749,203.708,-80.625,173.710,27.613,154.943
C06349=1071.755,203.957,-80.649,173.712,27.616,154.943
C06350=1071.760,204.206,-80.673,173.715,27.620,154.943
C06351=1071.766,204.455,-80.698,173.717,27.623,154.944
C06352=1071.772,204.703,-80.721,173.719,27.626,154.944
C06353=1071.777,204.951,-80.746,173.721,27.629,154.945
C06354=1071.783,205.201,-80.770,173.724,27.632,154.945
C06355=1071.788,205.449,-80.794,173.726,27.635,154.945
C06356=1071.794,205.698,-80.818,173.729,27.638,154.946
C06357=1071.800,205.947,-80.843,173.730,27.641,154.946
C06358=1071.806,206.196,-80.867,173.733,27.644,154.947
C06359=1071.811,206.444,-80.891,173.735,27.647,154.947
C06360=1071.817,206.693,-80.915,173.737,27.650,154.948
C06361=1071.841,207.735,-81.017,173.869,27.718,154.949
C06362=1071.851,208.156,-81.059,173.872,27.725,154.950
C06363=1071.861,208.576,-81.102,173.876,27.731,154.951
C06364=1071.871,208.997,-81.144,173.879,27.738,154.953
C06365=1071.880,209.418,-81.186,173.882,27.745,154.954
C06366=1071.886,209.667,-81.211,173.885,27.748,154.954
C06367=1071.892,209.916,-81.236,173.887,27.752,154.955
C06368=1071.898,210.164,-81.261,173.889,27.756,154.955
C06369=1071.904,210.412,-81.286,173.891,27.760,154.956
C06370=1071.910,210.661,-81.311,173.893,27.764,154.957
C06371=1071.916,210.910,-81.336,173.895,27.768,154.957
C06372=1071.921,211.159,-81.362,173.897,27.772,154.958
C06373=1071.927,211.407,-81.387,173.899,27.776,154.959
C06374=1071.933,211.657,-81.412,173.901,27.780,154.959
C06375=1071.939,211.905,-81.436,173.903,27.784,154.960
C06376=1071.945,212.153,-81.462,173.906,27.788,154.960
C06377=1071.951,212.402,-81.487,173.907,27.792,154.961
C06378=1071.956,212.651,-81.513,173.909,27.796,154.962
C06379=1071.962,212.900,-81.537,173.912,27.800,154.962
C06380=1071.968,213.148,-81.563,173.914,27.804,154.963
C06381=1071.974,213.397,-81.588,173.915,27.807,154.964
C06382=1071.979,213.645,-81.614,173.918,27.811,154.964
C06383=1071.985,213.894,-81.639,173.920,27.815,154.965
C06384=1071.991,214.142,-81.664,173.922,27.819,154.965
C06385=1071.997,214.391,-81.690,173.924,27.823,154.966
C06386=1072.002,214.640,-81.714,173.926,27.827,154.967
C06387=1072.008,214.889,-81.740,173.928,27.831,154.967
C06388=1072.014,215.138,-81.766,173.931,27.835,154.968
C06389=1072.020,215.386,-81.791,173.933,27.839,154.969
C06390=1072.026,215.634,-81.816,173.934,27.843,154.969
C06391=1072.031,215.883,-81.842,173.937,27.847,154.970
C06392=1072.037,216.132,-81.867,173.939,27.851,154.970
C06393=1072.044,216.381,-81.893,173.941,27.855,154.971
C06394=1072.049,216.630,-81.919,173.943,27.859,154.972
C06395=1072.055,216.878,-81.944,173.945,27.863,154.972
C06396=1072.061,217.126,-81.969,173.947,27.867,154.973
C06397=1072.066,217.375,-81.995,173.950,27.870,154.974
C06398=1072.073,217.624,-82.020,173.952,27.874,154.974
C06399=1072.078,217.873,-82.046,173.953,27.878,154.975
C06400=1072.084,218.121,-82.071,173.956,27.882,154.975
C06401=1072.090,218.370,-82.096,173.958,27.886,154.976
C06402=1072.095,218.619,-82.122,173.960,27.890,154.977
C06403=1072.101,218.867,-82.148,173.963,27.894,154.977
C06404=1072.108,219.115,-82.174,173.964,27.898,154.978
C06405=1072.113,219.364,-82.200,173.966,27.902,154.979
C06406=1072.120,219.613,-82.225,173.969,27.906,154.979
C06407=1072.125,219.862,-82.251,173.971,27.910,154.980
C06408=1072.131,220.110,-82.276,173.973,27.913,154.980
C06409=1072.136,220.359,-82.302,173.975,27.917,154.981
C06410=1072.142,220.607,-82.327,173.977,27.921,154.982
C06411=1072.149,220.856,-82.353,173.979,27.925,154.982
C06412=1072.154,221.104,-82.379,173.982,27.929,154.983
C06413=1072.161,221.353,-82.405,173.984,27.933,154.983
C06414=1072.165,221.566,-82.427,173.985,27.936,154.984
C06415=1072.171,221.778,-82.449,173.988,27.940,154.985
C06416=1072.175,221.991,-82.471,173.989,27.943,154.985
C06417=1072.180,222.204,-82.494,173.991,27.946,154.986
C06418=1072.186,222.416,-82.515,173.993,27.950,154.986
C06419=1072.190,222.628,-82.537,173.995,27.953,154.987
C06420=1072.195,222.841,-82.560,173.997,27.956,154.987
C06421=1072.200,223.054,-82.582,173.999,27.960,154.988
C06422=1072.206,223.303,-82.608,174.001,27.964,154.988
C06423=1072.212,223.551,-82.633,174.003,27.968,154.989
C06424=1072.218,223.800,-82.660,174.005,27.971,154.990
C06425=1072.223,224.049,-82.686,174.007,27.975,154.990
C06426=1072.229,224.297,-82.711,174.009,27.979,154.991
C06427=1072.235,224.546,-82.738,174.012,27.983,154.991
C06428=1072.241,224.795,-82.763,174.014,27.987,154.992
C06429=1072.247,225.043,-82.790,174.016,27.991,154.993
C06430=1072.253,225.292,-82.815,174.019,27.995,154.993
C06431=1072.258,225.541,-82.841,174.020,27.999,154.994
C06432=1072.264,225.788,-82.867,174.022,28.002,154.995
C06433=1072.269,226.037,-82.893,174.025,28.006,154.995
C06434=1072.275,226.285,-82.920,174.027,28.010,154.996
C06435=1072.281,226.534,-82.945,174.029,28.015,154.996
C06436=1072.287,226.782,-82.972,174.032,28.019,154.997
C06437=1072.293,227.031,-82.998,174.033,28.022,154.998
C06438=1072.299,227.280,-83.025,174.035,28.026,154.998
C06439=1072.305,227.529,-83.050,174.038,28.030,154.999
C06440=1072.311,227.777,-83.077,174.040,28.034,155.000
C06441=1072.316,228.026,-83.103,174.043,28.037,155.000
C06442=1072.323,228.274,-83.129,174.045,28.041,155.001
C06443=1072.328,228.523,-83.155,174.047,28.046,155.001
C06444=1072.334,228.772,-83.181,174.050,28.050,155.002
C06445=1072.340,229.020,-83.208,174.051,28.053,155.003
C06446=1072.346,229.269,-83.233,174.053,28.057,155.003
C06447=1072.352,229.517,-83.260,174.056,28.061,155.004
C06448=1072.358,229.765,-83.286,174.058,28.065,155.004
C06449=1072.363,230.014,-83.312,174.060,28.068,155.005
C06450=1072.370,230.263,-83.338,174.063,28.072,155.006
C06451=1072.376,230.511,-83.365,174.065,28.076,155.006
C06452=1072.381,230.760,-83.391,174.067,28.080,155.007
C06453=1072.387,231.008,-83.418,174.069,28.084,155.008
C06454=1072.393,231.257,-83.445,174.071,28.088,155.008
C06455=1072.399,231.506,-83.471,174.074,28.092,155.009
C06456=1072.404,231.755,-83.497,174.076,28.096,155.009
C06457=1072.410,232.003,-83.524,174.078,28.100,155.010
C06458=1072.416,232.251,-83.551,174.081,28.104,155.011
C06459=1072.421,232.500,-83.576,174.083,28.108,155.011
C06460=1072.427,232.749,-83.603,174.085,28.111,155.012
C06461=1072.433,232.997,-83.630,174.088,28.115,155.012
C06462=1072.439,233.245,-83.656,174.089,28.119,155.013
C06463=1072.446,233.494,-83.683,174.091,28.123,155.014
C06464=1072.452,233.743,-83.709,174.094,28.127,155.014
C06465=1072.457,233.991,-83.735,174.096,28.131,155.015
C06466=1072.462,234.240,-83.763,174.099,28.135,155.016
C06467=1072.468,234.489,-83.789,174.101,28.139,155.016
C06468=1072.474,234.737,-83.816,174.103,28.143,155.017
C06469=1072.479,234.985,-83.843,174.106,28.147,155.017
C06470=1072.489,235.402,-83.887,174.110,28.153,155.018
C06471=1072.499,235.819,-83.932,174.114,28.160,155.020
C06472=1072.509,236.236,-83.977,174.116,28.166,155.021
C06473=1072.519,236.653,-84.022,174.120,28.173,155.022
C06474=1072.525,236.902,-84.049,174.123,28.176,155.022
C06475=1072.531,237.150,-84.075,174.125,28.180,155.023
C06476=1072.537,237.398,-84.102,174.128,28.184,155.023
C06477=1072.542,237.647,-84.129,174.130,28.188,155.024
C06478=1072.548,237.896,-84.156,174.132,28.192,155.025
C06479=1072.554,238.145,-84.183,174.135,28.196,155.025
C06480=1072.560,238.393,-84.210,174.137,28.200,155.026
C06481=1072.565,238.641,-84.236,174.139,28.204,155.027
C06482=1072.572,238.890,-84.263,174.142,28.208,155.027
C06483=1072.578,239.139,-84.290,174.144,28.211,155.028
C06484=1072.584,239.386,-84.317,174.147,28.215,155.028
C06485=1072.589,239.635,-84.344,174.149,28.219,155.029
C06486=1072.595,239.884,-84.372,174.151,28.223,155.030
C06487=1072.601,240.132,-84.398,174.154,28.227,155.030
C06488=1072.607,240.381,-84.425,174.155,28.231,155.031
C06489=1072.613,240.629,-84.452,174.157,28.235,155.031
C06490=1072.619,240.878,-84.479,174.160,28.239,155.032
C06491=1072.624,241.126,-84.507,174.162,28.243,155.033
C06492=1072.630,241.375,-84.533,174.165,28.246,155.033
C06493=1072.636,241.624,-84.560,174.167,28.250,155.034
C06494=1072.642,241.871,-84.588,174.169,28.254,155.035
C06495=1072.648,242.120,-84.614,174.172,28.258,155.035
C06496=1072.654,242.369,-84.642,174.174,28.262,155.036
C06497=1072.660,242.617,-84.669,174.176,28.266,155.036
C06498=1072.666,242.865,-84.696,174.179,28.270,155.037
C06499=1072.671,243.114,-84.723,174.181,28.274,155.038
C06500=1072.677,243.362,-84.751,174.184,28.277,155.038
C06501=1072.683,243.611,-84.777,174.186,28.281,155.039
C06502=1072.688,243.859,-84.805,174.188,28.285,155.039
C06503=1072.695,244.108,-84.832,174.191,28.289,155.040
C06504=1072.700,244.357,-84.860,174.193,28.293,155.041
C06505=1072.706,244.604,-84.887,174.195,28.297,155.041
C06506=1072.712,244.853,-84.914,174.198,28.301,155.042
C06507=1072.718,245.101,-84.942,174.200,28.305,155.043
C06508=1072.723,245.350,-84.969,174.203,28.309,155.043
C06509=1072.729,245.599,-84.997,174.205,28.313,155.044
C06510=1072.735,245.847,-85.024,174.207,28.317,155.044
C06511=1072.741,246.095,-85.050,174.210,28.320,155.045
C06512=1072.747,246.344,-85.079,174.212,28.324,155.046
C06513=1072.753,246.592,-85.106,174.215,28.328,155.046
C06514=1072.759,246.841,-85.134,174.217,28.332,155.047
C06515=1072.765,247.089,-85.161,174.219,28.336,155.048
C06516=1072.770,247.338,-85.188,174.222,28.340,155.048
C06517=1072.776,247.586,-85.216,174.224,28.344,155.049
C06518=1072.781,247.835,-85.243,174.227,28.348,155.049
C06519=1072.787,248.083,-85.271,174.229,28.352,155.050
C06520=1072.793,248.331,-85.299,174.231,28.356,155.051
C06521=1072.798,248.580,-85.326,174.234,28.360,155.051
C06522=1072.807,248.974,-85.370,174.238,28.366,155.052
C06523=1072.817,249.369,-85.415,174.241,28.372,155.053
C06524=1072.826,249.763,-85.459,174.245,28.378,155.054
C06525=1072.835,250.157,-85.502,174.249,28.385,155.055
C06526=1072.840,250.406,-85.530,174.251,28.388,155.056
C06527=1072.847,250.654,-85.558,174.254,28.392,155.057
C06528=1072.852,250.902,-85.586,174.256,28.396,155.057
C06529=1072.858,251.151,-85.613,174.258,28.400,155.058
C06530=1072.864,251.399,-85.641,174.261,28.404,155.059
C06531=1072.870,251.648,-85.669,174.263,28.408,155.059
C06532=1072.875,251.896,-85.697,174.265,28.412,155.060
C06533=1072.882,252.144,-85.725,174.268,28.416,155.060
C06534=1072.887,252.392,-85.752,174.270,28.420,155.061
C06535=1072.893,252.642,-85.780,174.273,28.424,155.062
C06536=1072.899,252.889,-85.807,174.275,28.428,155.062
C06537=1072.905,253.138,-85.836,174.277,28.432,155.063
C06538=1072.910,253.386,-85.864,174.280,28.436,155.064
C06539=1072.916,253.635,-85.892,174.282,28.439,155.064
C06540=1072.922,253.883,-85.919,174.285,28.443,155.065
C06541=1072.928,254.132,-85.948,174.288,28.447,155.065
C06542=1072.933,254.380,-85.976,174.290,28.451,155.066
C06543=1072.939,254.628,-86.004,174.293,28.455,155.067
C06544=1072.945,254.876,-86.031,174.295,28.459,155.067
C06545=1072.951,255.125,-86.060,174.298,28.463,155.068
C06546=1072.957,255.373,-86.088,174.300,28.467,155.068
C06547=1072.963,255.622,-86.116,174.302,28.471,155.069
C06548=1072.969,255.870,-86.144,174.305,28.475,155.070
C06549=1072.975,256.118,-86.172,174.307,28.479,155.070
C06550=1072.980,256.367,-86.200,174.310,28.482,155.071
C06551=1072.986,256.615,-86.228,174.312,28.486,155.072
C06552=1072.993,256.863,-86.256,174.314,28.490,155.072
C06553=1072.998,257.112,-86.284,174.317,28.494,155.073
C06554=1073.004,257.360,-86.312,174.319,28.498,155.073
C06555=1073.010,257.609,-86.340,174.322,28.502,155.074
C06556=1073.016,257.857,-86.369,174.325,28.506,155.075
C06557=1073.022,258.105,-86.397,174.328,28.510,155.075
C06558=1073.028,258.354,-86.425,174.330,28.514,155.076
C06559=1073.034,258.602,-86.453,174.332,28.517,155.076
C06560=1073.039,258.850,-86.481,174.335,28.521,155.077
C06561=1073.045,259.099,-86.510,174.337,28.525,155.078
C06562=1073.052,259.347,-86.538,174.340,28.529,155.078
C06563=1073.058,259.595,-86.566,174.342,28.533,155.079
C06564=1073.064,259.844,-86.594,174.344,28.537,155.080
C06565=1073.069,260.092,-86.623,174.347,28.541,155.080
C06566=1073.076,260.356,-86.653,174.350,28.545,155.081
C06567=1073.083,260.621,-86.683,174.353,28.549,155.081
C06568=1073.089,260.885,-86.713,174.355,28.553,155.082
C06569=1073.095,261.150,-86.744,174.358,28.557,155.083
C06570=1073.101,261.398,-86.771,174.361,28.561,155.083
C06571=1073.107,261.645,-86.800,174.363,28.565,155.084
C06572=1073.113,261.894,-86.828,174.366,28.569,155.085
C06573=1073.119,262.143,-86.857,174.368,28.572,155.085
C06574=1073.129,262.550,-86.904,174.372,28.579,155.086
C06575=1073.139,262.959,-86.951,174.376,28.585,155.087
C06576=1073.149,263.366,-86.997,174.381,28.592,155.088
C06577=1073.159,263.774,-87.044,174.385,28.598,155.089
C06578=1073.165,264.022,-87.072,174.388,28.602,155.090
C06579=1073.171,264.270,-87.101,174.390,28.606,155.091
C06580=1073.176,264.520,-87.130,174.392,28.610,155.091
C06581=1073.182,264.767,-87.159,174.395,28.614,155.092
C06582=1073.188,265.016,-87.187,174.397,28.618,155.093
C06583=1073.194,265.264,-87.216,174.401,28.621,155.093
C06584=1073.200,265.513,-87.245,174.403,28.625,155.094
C06585=1073.205,265.760,-87.273,174.406,28.629,155.094
C06586=1073.212,266.008,-87.302,174.408,28.633,155.095
C06587=1073.217,266.257,-87.331,174.410,28.637,155.096
C06588=1073.223,266.505,-87.360,174.413,28.641,155.096
C06589=1073.229,266.753,-87.388,174.415,28.645,155.097
C06590=1073.235,267.002,-87.417,174.419,28.649,155.098
C06591=1073.241,267.250,-87.446,174.421,28.653,155.098
C06592=1073.246,267.499,-87.475,174.423,28.657,155.099
C06593=1073.252,267.747,-87.504,174.426,28.661,155.099
C06594=1073.259,267.995,-87.533,174.428,28.665,155.100
C06595=1073.264,268.242,-87.562,174.431,28.669,155.101
C06596=1073.270,268.491,-87.590,174.434,28.673,155.101
C06597=1073.276,268.740,-87.620,174.436,28.677,155.102
C06598=1073.282,268.988,-87.649,174.439,28.681,155.103
C06599=1073.288,269.236,-87.678,174.441,28.685,155.103
C06600=1073.294,269.485,-87.706,174.444,28.689,155.104
C06601=1073.300,269.733,-87.736,174.446,28.693,155.105
C06602=1073.305,269.981,-87.765,174.450,28.696,155.105
C06603=1073.312,270.229,-87.794,174.452,28.700,155.106
C06604=1073.317,270.477,-87.823,174.454,28.704,155.106
C06605=1073.323,270.725,-87.852,174.457,28.708,155.107
C06606=1073.329,270.974,-87.881,174.459,28.712,155.108
C06607=1073.335,271.222,-87.910,174.462,28.716,155.108
C06608=1073.341,271.471,-87.939,174.465,28.720,155.109
C06609=1073.347,271.719,-87.969,174.468,28.724,155.110
C06610=1073.352,271.966,-87.998,174.470,28.728,155.110
C06611=1073.359,272.215,-88.027,174.472,28.732,155.111
C06612=1073.364,272.463,-88.056,174.475,28.736,155.112
C06613=1073.370,272.711,-88.086,174.478,28.740,155.112
C06614=1073.377,272.959,-88.115,174.481,28.744,155.113
C06615=1073.382,273.208,-88.144,174.483,28.748,155.113
C06616=1073.388,273.456,-88.173,174.486,28.752,155.114
C06617=1073.394,273.704,-88.203,174.488,28.756,155.115
C06618=1073.400,273.952,-88.232,174.491,28.760,155.115
C06619=1073.406,274.201,-88.262,174.494,28.764,155.116
C06620=1073.412,274.449,-88.291,174.496,28.768,155.117
C06621=1073.417,274.697,-88.320,174.499,28.772,155.117
C06622=1073.424,274.945,-88.350,174.501,28.776,155.118
C06623=1073.429,275.193,-88.380,174.504,28.780,155.119
C06624=1073.436,275.442,-88.409,174.507,28.784,155.119
C06625=1073.441,275.690,-88.438,174.509,28.788,155.120
C06626=1073.451,276.101,-88.487,174.513,28.794,155.121
C06627=1073.460,276.512,-88.536,174.518,28.801,155.122
C06628=1073.470,276.923,-88.585,174.523,28.808,155.123
C06629=1073.480,277.334,-88.634,174.528,28.814,155.124
C06630=1073.486,277.582,-88.663,174.530,28.818,155.125
C06631=1073.492,277.830,-88.693,174.532,28.822,155.125
C06632=1073.497,278.079,-88.723,174.535,28.826,155.126
C06633=1073.503,278.327,-88.752,174.538,28.830,155.127
C06634=1073.509,278.575,-88.782,174.541,28.834,155.127
C06635=1073.516,278.823,-88.811,174.543,28.838,155.128
C06636=1073.521,279.071,-88.841,174.546,28.842,155.129
C06637=1073.527,279.320,-88.872,174.549,28.846,155.129
C06638=1073.534,279.568,-88.901,174.551,28.850,155.130
C06639=1073.539,279.816,-88.930,174.554,28.855,155.131
C06640=1073.545,280.064,-88.961,174.556,28.859,155.131
C06641=1073.551,280.312,-88.990,174.560,28.863,155.132
C06642=1073.557,280.560,-89.020,174.562,28.867,155.133
C06643=1073.563,280.808,-89.050,174.565,28.871,155.133
C06644=1073.569,281.056,-89.079,174.567,28.875,155.134
C06645=1073.575,281.304,-89.109,174.570,28.879,155.135
C06646=1073.581,281.552,-89.139,174.573,28.883,155.135
C06647=1073.586,281.801,-89.169,174.575,28.887,155.136
C06648=1073.592,282.048,-89.199,174.578,28.891,155.137
C06649=1073.598,282.298,-89.229,174.581,28.895,155.137
C06650=1073.604,282.545,-89.260,174.584,28.899,155.138
C06651=1073.610,282.793,-89.289,174.586,28.903,155.139
C06652=1073.616,283.041,-89.319,174.589,28.907,155.139
C06653=1073.622,283.289,-89.349,174.592,28.911,155.140
C06654=1073.627,283.538,-89.379,174.594,28.915,155.141
C06655=1073.633,283.785,-89.409,174.597,28.919,155.141
C06656=1073.639,284.033,-89.440,174.600,28.923,155.142
C06657=1073.644,284.282,-89.469,174.603,28.927,155.142
C06658=1073.651,284.530,-89.500,174.605,28.932,155.143
C06659=1073.657,284.778,-89.530,174.608,28.936,155.144
C06660=1073.663,285.026,-89.560,174.611,28.940,155.145
C06661=1073.669,285.274,-89.590,174.613,28.944,155.145
C06662=1073.674,285.522,-89.620,174.616,28.947,155.146
C06663=1073.681,285.770,-89.651,174.619,28.952,155.146
C06664=1073.686,286.019,-89.681,174.622,28.956,155.147
C06665=1073.692,286.267,-89.711,174.624,28.960,155.148
C06666=1073.698,286.514,-89.741,174.627,28.964,155.149
C06667=1073.704,286.762,-89.772,174.630,28.968,155.149
C06668=1073.711,287.010,-89.802,174.632,28.972,155.150
C06669=1073.717,287.258,-89.832,174.636,28.976,155.150
C06670=1073.722,287.507,-89.862,174.638,28.980,155.151
C06671=1073.728,287.755,-89.892,174.641,28.984,155.152
C06672=1073.735,288.003,-89.923,174.644,28.988,155.152
C06673=1073.740,288.251,-89.953,174.647,28.993,155.153
C06674=1073.746,288.499,-89.984,174.649,28.997,155.154
C06675=1073.752,288.747,-90.014,174.652,29.001,155.155
C06676=1073.758,288.995,-90.045,174.655,29.005,155.155
C06677=1073.764,289.243,-90.075,174.657,29.008,155.156
C06678=1073.769,289.453,-90.101,174.660,29.012,155.156
C06679=1073.775,289.664,-90.127,174.662,29.016,155.157
C06680=1073.779,289.875,-90.153,174.665,29.019,155.158
C06681=1073.784,290.085,-90.179,174.667,29.023,155.158
C06682=1073.789,290.296,-90.205,174.669,29.026,155.159
C06683=1073.795,290.507,-90.230,174.671,29.030,155.159
C06684=1073.799,290.718,-90.256,174.674,29.033,155.160
C06685=1073.804,290.928,-90.282,174.676,29.037,155.160
C06686=1073.810,291.176,-90.313,174.679,29.041,155.161
C06687=1073.816,291.424,-90.344,174.682,29.045,155.162
C06688=1073.822,291.671,-90.374,174.685,29.049,155.162
C06689=1073.829,291.920,-90.405,174.687,29.053,155.163
C06690=1073.834,292.168,-90.436,174.691,29.057,155.164
C06691=1073.839,292.416,-90.466,174.693,29.061,155.165
C06692=1073.846,292.664,-90.497,174.696,29.066,155.165
C06693=1073.852,292.912,-90.528,174.699,29.070,155.166
C06694=1073.858,293.160,-90.558,174.701,29.074,155.167
C06695=1073.864,293.408,-90.590,174.705,29.078,155.167
C06696=1073.869,293.656,-90.620,174.707,29.082,155.168
C06697=1073.876,293.905,-90.651,174.710,29.086,155.169
C06698=1073.882,294.152,-90.682,174.713,29.090,155.169
C06699=1073.888,294.400,-90.712,174.716,29.095,155.170
C06700=1073.893,294.649,-90.743,174.719,29.099,155.171
C06701=1073.899,294.896,-90.775,174.722,29.103,155.171
C06702=1073.905,295.144,-90.805,174.724,29.107,155.172
C06703=1073.912,295.392,-90.836,174.727,29.111,155.173
C06704=1073.917,295.640,-90.867,174.730,29.115,155.173
C06705=1073.924,295.888,-90.898,174.733,29.120,155.174
C06706=1073.930,296.135,-90.929,174.736,29.124,155.175
C06707=1073.935,296.384,-90.960,174.738,29.128,155.176
C06708=1073.941,296.632,-90.991,174.742,29.132,155.176
C06709=1073.947,296.879,-91.022,174.744,29.136,155.177
C06710=1073.953,297.128,-91.053,174.747,29.140,155.178
C06711=1073.959,297.375,-91.084,174.750,29.145,155.178
C06712=1073.965,297.624,-91.115,174.752,29.149,155.179
C06713=1073.971,297.871,-91.147,174.756,29.153,155.180
C06714=1073.977,298.120,-91.178,174.758,29.157,155.180
C06715=1073.983,298.367,-91.209,174.762,29.162,155.181
C06716=1073.988,298.615,-91.240,174.764,29.166,155.182
C06717=1073.994,298.864,-91.272,174.767,29.170,155.183
C06718=1074.000,299.111,-91.303,174.770,29.175,155.183
C06719=1074.006,299.360,-91.334,174.772,29.179,155.184
C06720=1074.012,299.607,-91.365,174.776,29.183,155.185
C06721=1074.017,299.854,-91.397,174.778,29.187,155.185
C06722=1074.023,300.103,-91.428,174.782,29.192,155.186
C06723=1074.029,300.350,-91.459,174.784,29.196,155.187
C06724=1074.035,300.599,-91.491,174.787,29.200,155.188
C06725=1074.041,300.846,-91.522,174.790,29.205,155.188
C06726=1074.047,301.095,-91.554,174.792,29.209,155.189
C06727=1074.052,301.342,-91.585,174.796,29.213,155.190
C06728=1074.059,301.590,-91.617,174.798,29.217,155.191
C06729=1074.064,301.838,-91.648,174.802,29.222,155.191
C06730=1074.070,302.086,-91.680,174.804,29.226,155.192
C06731=1074.076,302.334,-91.711,174.808,29.231,155.193
C06732=1074.082,302.582,-91.743,174.810,29.235,155.193
C06733=1074.087,302.829,-91.775,174.814,29.239,155.194
C06734=1074.093,303.048,-91.802,174.816,29.243,155.195
C06735=1074.098,303.266,-91.830,174.819,29.247,155.195
C06736=1074.103,303.483,-91.857,174.821,29.251,155.196
C06737=1074.108,303.702,-91.885,174.824,29.255,155.197
C06738=1074.113,303.919,-91.913,174.826,29.258,155.197
C06739=1074.119,304.138,-91.941,174.829,29.262,155.198
C06740=1074.124,304.355,-91.969,174.831,29.266,155.199
C06741=1074.129,304.574,-91.997,174.834,29.270,155.199
C06742=1074.135,304.821,-92.028,174.836,29.273,155.200
C06743=1074.141,305.069,-92.060,174.839,29.278,155.201
C06744=1074.147,305.317,-92.092,174.842,29.282,155.202
C06745=1074.153,305.565,-92.123,174.845,29.287,155.202
C06746=1074.159,305.813,-92.155,174.848,29.291,155.203
C06747=1074.165,306.060,-92.186,174.851,29.296,155.204
C06748=1074.171,306.309,-92.218,174.854,29.299,155.204
C06749=1074.177,306.556,-92.250,174.857,29.304,155.205
C06750=1074.183,306.803,-92.282,174.860,29.309,155.206
C06751=1074.189,307.052,-92.314,174.863,29.313,155.207
C06752=1074.195,307.300,-92.346,174.865,29.317,155.207
C06753=1074.202,307.548,-92.378,174.869,29.322,155.208
C06754=1074.207,307.795,-92.409,174.871,29.326,155.209
C06755=1074.213,308.043,-92.441,174.875,29.330,155.210
C06756=1074.219,308.292,-92.473,174.878,29.334,155.210
C06757=1074.226,308.538,-92.505,174.881,29.339,155.211
C06758=1074.232,308.786,-92.537,174.884,29.343,155.212
C06759=1074.237,309.035,-92.569,174.887,29.348,155.212
C06760=1074.243,309.283,-92.601,174.890,29.352,155.213
C06761=1074.249,309.530,-92.633,174.893,29.356,155.214
C06762=1074.256,309.778,-92.665,174.896,29.361,155.215
C06763=1074.262,310.026,-92.697,174.898,29.365,155.215
C06764=1074.268,310.274,-92.729,174.902,29.369,155.216
C06765=1074.274,310.522,-92.762,174.904,29.374,155.217
C06766=1074.280,310.769,-92.794,174.908,29.378,155.218
C06767=1074.286,311.017,-92.825,174.910,29.382,155.218
C06768=1074.293,311.265,-92.858,174.914,29.387,155.219
C06769=1074.299,311.513,-92.890,174.917,29.391,155.220
C06770=1074.305,311.761,-92.922,174.920,29.395,155.221
C06771=1074.311,312.009,-92.955,174.923,29.400,155.221
C06772=1074.316,312.256,-92.986,174.925,29.404,155.222
C06773=1074.323,312.504,-93.019,174.929,29.408,155.223
C06774=1074.329,312.752,-93.050,174.931,29.413,155.224
C06775=1074.335,313.000,-93.082,174.935,29.417,155.224
C06776=1074.342,313.247,-93.115,174.937,29.422,155.225
C06777=1074.348,313.496,-93.147,174.941,29.426,155.226
C06778=1074.354,313.743,-93.180,174.944,29.430,155.226
C06779=1074.360,313.992,-93.212,174.947,29.435,155.227
C06780=1074.366,314.239,-93.245,174.950,29.439,155.228
C06781=1074.372,314.487,-93.277,174.953,29.443,155.229
C06782=1074.378,314.734,-93.309,174.956,29.448,155.229
C06783=1074.384,314.982,-93.342,174.958,29.453,155.230
C06784=1074.390,315.230,-93.374,174.962,29.457,155.231
C06785=1074.396,315.478,-93.407,174.965,29.462,155.232
C06786=1074.402,315.726,-93.440,174.968,29.466,155.233
C06787=1074.408,315.974,-93.472,174.971,29.471,155.233
C06788=1074.413,316.221,-93.505,174.974,29.475,155.234
C06789=1074.419,316.469,-93.538,174.977,29.480,155.235
C06790=1074.424,316.689,-93.566,174.980,29.484,155.236
C06791=1074.430,316.908,-93.595,174.982,29.488,155.236
C06792=1074.435,317.128,-93.624,174.985,29.492,155.237
C06793=1074.440,317.348,-93.654,174.988,29.496,155.238
C06794=1074.445,317.567,-93.683,174.991,29.500,155.239
C06795=1074.451,317.787,-93.711,174.993,29.504,155.239
C06796=1074.456,318.006,-93.741,174.996,29.508,155.240
C06797=1074.461,318.225,-93.770,174.998,29.512,155.241
C06798=1074.467,318.474,-93.802,175.002,29.517,155.241
C06799=1074.474,318.721,-93.835,175.005,29.522,155.242
C06800=1074.479,318.969,-93.868,175.008,29.526,155.243
C06801=1074.485,319.217,-93.901,175.011,29.531,155.244
C06802=1074.491,319.465,-93.935,175.013,29.535,155.245
C06803=1074.497,319.712,-93.967,175.017,29.540,155.245
C06804=1074.503,319.960,-94.000,175.020,29.545,155.246
C06805=1074.509,320.208,-94.033,175.023,29.549,155.247
C06806=1074.515,320.455,-94.066,175.026,29.554,155.248
C06807=1074.521,320.703,-94.099,175.030,29.559,155.249
C06808=1074.527,320.951,-94.132,175.032,29.563,155.249
C06809=1074.533,321.198,-94.165,175.036,29.568,155.250
C06810=1074.539,321.446,-94.198,175.038,29.572,155.251
C06811=1074.545,321.694,-94.231,175.041,29.577,155.252
C06812=1074.551,321.942,-94.264,175.045,29.582,155.253
C06813=1074.557,322.189,-94.297,175.047,29.586,155.253
C06814=1074.563,322.437,-94.330,175.051,29.591,155.254
C06815=1074.569,322.685,-94.363,175.054,29.596,155.255
C06816=1074.575,322.932,-94.396,175.057,29.600,155.256
C06817=1074.581,323.180,-94.429,175.060,29.605,155.257
C06818=1074.587,323.428,-94.462,175.064,29.609,155.257
C06819=1074.594,323.676,-94.496,175.066,29.614,155.258
C06820=1074.600,323.924,-94.529,175.070,29.619,155.259
C06821=1074.605,324.171,-94.563,175.073,29.623,155.260
C06822=1074.612,324.419,-94.595,175.075,29.628,155.261
C06823=1074.617,324.667,-94.629,175.079,29.633,155.262
C06824=1074.624,324.914,-94.662,175.082,29.637,155.262
C06825=1074.630,325.163,-94.696,175.085,29.642,155.263
C06826=1074.636,325.410,-94.729,175.088,29.647,155.264
C06827=1074.642,325.657,-94.763,175.092,29.651,155.265
C06828=1074.649,325.905,-94.795,175.094,29.656,155.266
C06829=1074.654,326.153,-94.829,175.098,29.661,155.267
C06830=1074.661,326.401,-94.862,175.101,29.665,155.267
C06831=1074.667,326.648,-94.896,175.104,29.670,155.268
C06832=1074.673,326.896,-94.929,175.107,29.675,155.269
C06833=1074.679,327.143,-94.963,175.110,29.680,155.270
C06834=1074.686,327.392,-94.996,175.114,29.684,155.271
C06835=1074.692,327.639,-95.030,175.116,29.689,155.271
C06836=1074.697,327.887,-95.063,175.120,29.694,155.272
C06837=1074.704,328.134,-95.096,175.123,29.698,155.273
C06838=1074.710,328.382,-95.130,175.127,29.704,155.274
C06839=1074.716,328.630,-95.163,175.129,29.708,155.275
C06840=1074.722,328.877,-95.197,175.133,29.712,155.276
C06841=1074.729,329.126,-95.230,175.136,29.718,155.276
C06842=1074.735,329.373,-95.264,175.139,29.722,155.277
C06843=1074.741,329.620,-95.298,175.142,29.727,155.278
C06844=1074.748,329.868,-95.331,175.145,29.732,155.279
C06845=1074.754,330.116,-95.365,175.149,29.737,155.280
C06846=1074.759,330.332,-95.395,175.151,29.740,155.281
C06847=1074.765,330.548,-95.424,175.154,29.745,155.281
C06848=1074.771,330.765,-95.454,175.157,29.749,155.282
C06849=1074.776,330.982,-95.483,175.160,29.753,155.283
C06850=1074.781,331.198,-95.513,175.162,29.757,155.284
C06851=1074.787,331.414,-95.543,175.165,29.761,155.284
C06852=1074.792,331.631,-95.572,175.169,29.766,155.285
C06853=1074.797,331.847,-95.602,175.171,29.770,155.286
C06854=1074.803,332.095,-95.635,175.174,29.775,155.287
C06855=1074.810,332.343,-95.669,175.178,29.780,155.287
C06856=1074.816,332.590,-95.703,175.180,29.785,155.288
C06857=1074.822,332.837,-95.737,175.184,29.790,155.289
C06858=1074.828,333.085,-95.771,175.187,29.795,155.290
C06859=1074.834,333.332,-95.805,175.191,29.800,155.291
C06860=1074.839,333.580,-95.839,175.193,29.804,155.292
C06861=1074.846,333.828,-95.873,175.197,29.809,155.293
C06862=1074.852,334.076,-95.907,175.200,29.814,155.294
C06863=1074.858,334.324,-95.942,175.204,29.819,155.295
C06864=1074.864,334.571,-95.976,175.207,29.824,155.295
C06865=1074.871,334.819,-96.010,175.209,29.829,155.296
C06866=1074.876,335.066,-96.044,175.213,29.834,155.297
C06867=1074.882,335.313,-96.078,175.216,29.839,155.298
C06868=1074.889,335.561,-96.113,175.220,29.844,155.299
C06869=1074.895,335.809,-96.147,175.223,29.849,155.300
C06870=1074.901,336.057,-96.181,175.226,29.854,155.301
C06871=1074.907,336.304,-96.215,175.229,29.859,155.302
C06872=1074.913,336.552,-96.250,175.233,29.864,155.303
C06873=1074.919,336.799,-96.284,175.236,29.869,155.303
C06874=1074.926,337.047,-96.318,175.240,29.874,155.304
C06875=1074.932,337.295,-96.352,175.243,29.879,155.305
C06876=1074.938,337.542,-96.387,175.245,29.884,155.306
C06877=1074.944,337.789,-96.421,175.249,29.889,155.307
C06878=1074.951,338.037,-96.456,175.252,29.894,155.308
C06879=1074.957,338.284,-96.490,175.256,29.899,155.309
C06880=1074.963,338.532,-96.524,175.259,29.904,155.310
C06881=1074.969,338.779,-96.559,175.263,29.909,155.311
C06882=1074.975,339.027,-96.594,175.265,29.914,155.312
C06883=1074.981,339.275,-96.628,175.269,29.920,155.313
C06884=1074.987,339.523,-96.662,175.272,29.925,155.314
C06885=1074.994,339.770,-96.698,175.276,29.930,155.314
C06886=1075.000,340.017,-96.732,175.279,29.935,155.315
C06887=1075.006,340.266,-96.767,175.282,29.940,155.316
C06888=1075.012,340.512,-96.801,175.286,29.945,155.317
C06889=1075.018,340.760,-96.836,175.288,29.950,155.318
C06890=1075.024,341.007,-96.871,175.292,29.955,155.319
C06891=1075.030,341.255,-96.906,175.295,29.960,155.320
C06892=1075.037,341.503,-96.940,175.299,29.966,155.321
C06893=1075.043,341.750,-96.975,175.302,29.971,155.322
C06894=1075.049,341.998,-97.009,175.306,29.976,155.323
C06895=1075.055,342.246,-97.045,175.309,29.981,155.324
C06896=1075.061,342.493,-97.079,175.313,29.986,155.325
C06897=1075.068,342.740,-97.114,175.316,29.992,155.326
C06898=1075.074,342.988,-97.149,175.318,29.996,155.327
C06899=1075.080,343.235,-97.184,175.322,30.002,155.328
C06900=1075.086,343.483,-97.219,175.325,30.007,155.329
C06901=1075.093,343.731,-97.253,175.329,30.012,155.329
C06902=1075.098,343.944,-97.284,175.332,30.017,155.330
C06903=1075.104,344.158,-97.314,175.335,30.021,155.331
C06904=1075.109,344.371,-97.345,175.337,30.026,155.332
C06905=1075.114,344.585,-97.374,175.341,30.031,155.333
C06906=1075.119,344.799,-97.405,175.343,30.035,155.334
C06907=1075.125,345.013,-97.435,175.346,30.039,155.334
C06908=1075.130,345.227,-97.465,175.350,30.044,155.335
C06909=1075.135,345.440,-97.496,175.352,30.049,155.336
C06910=1075.142,345.688,-97.531,175.355,30.054,155.337
C06911=1075.148,345.936,-97.566,175.359,30.059,155.338
C06912=1075.154,346.182,-97.601,175.362,30.065,155.339
C06913=1075.160,346.430,-97.637,175.366,30.070,155.340
C06914=1075.167,346.677,-97.672,175.369,30.075,155.341
C06915=1075.172,346.926,-97.707,175.373,30.081,155.342
C06916=1075.178,347.172,-97.742,175.376,30.086,155.343
C06917=1075.184,347.420,-97.778,175.380,30.091,155.344
C06918=1075.191,347.667,-97.813,175.383,30.097,155.345
C06919=1075.197,347.915,-97.848,175.387,30.102,155.346
C06920=1075.203,348.162,-97.883,175.390,30.107,155.347
C06921=1075.209,348.409,-97.919,175.394,30.113,155.348
C06922=1075.216,348.657,-97.954,175.397,30.118,155.349
C06923=1075.222,348.904,-97.990,175.400,30.124,155.350
C06924=1075.228,349.152,-98.026,175.404,30.129,155.351
C06925=1075.235,349.399,-98.061,175.407,30.134,155.352
C06926=1075.241,349.646,-98.096,175.411,30.140,155.353
C06927=1075.247,349.894,-98.131,175.414,30.146,155.354
C06928=1075.253,350.141,-98.167,175.418,30.151,155.355
C06929=1075.259,350.389,-98.203,175.421,30.157,155.356
C06930=1075.266,350.636,-98.238,175.425,30.162,155.357
C06931=1075.272,350.884,-98.274,175.428,30.167,155.358
C06932=1075.278,351.131,-98.310,175.432,30.173,155.359
C06933=1075.285,351.378,-98.345,175.435,30.178,155.360
C06934=1075.291,351.626,-98.380,175.438,30.184,155.361
C06935=1075.297,351.873,-98.416,175.442,30.189,155.362
C06936=1075.304,352.120,-98.452,175.445,30.195,155.363
C06937=1075.310,352.368,-98.488,175.449,30.200,155.364
C06938=1075.316,352.615,-98.523,175.452,30.206,155.365
C06939=1075.322,352.862,-98.560,175.456,30.211,155.366
C06940=1075.329,353.110,-98.595,175.459,30.217,155.367
C06941=1075.335,353.357,-98.631,175.463,30.223,155.369
C06942=1075.341,353.604,-98.667,175.466,30.228,155.370
C06943=1075.347,353.852,-98.703,175.470,30.234,155.371
C06944=1075.353,354.100,-98.739,175.473,30.239,155.372
C06945=1075.360,354.347,-98.775,175.476,30.245,155.373
C06946=1075.366,354.594,-98.810,175.480,30.251,155.374
C06947=1075.373,354.841,-98.847,175.483,30.256,155.375
C06948=1075.379,355.089,-98.882,175.487,30.262,155.376
C06949=1075.385,355.336,-98.919,175.490,30.268,155.377
C06950=1075.391,355.584,-98.955,175.494,30.273,155.378
C06951=1075.398,355.831,-98.991,175.497,30.279,155.379
C06952=1075.404,356.078,-99.027,175.501,30.285,155.380
C06953=1075.410,356.325,-99.063,175.505,30.291,155.381
C06954=1075.416,356.573,-99.100,175.509,30.296,155.382
C06955=1075.422,356.820,-99.135,175.512,30.302,155.383
C06956=1075.429,357.067,-99.171,175.516,30.308,155.385
C06957=1075.436,357.314,-99.208,175.519,30.314,155.386
C06958=1075.441,357.529,-99.239,175.522,30.318,155.387
C06959=1075.446,357.745,-99.271,175.525,30.323,155.388
C06960=1075.452,357.961,-99.303,175.529,30.328,155.388
C06961=1075.458,358.176,-99.334,175.531,30.334,155.389
C06962=1075.463,358.392,-99.365,175.535,30.339,155.390
C06963=1075.468,358.607,-99.397,175.537,30.343,155.391
C06964=1075.474,358.823,-99.429,175.541,30.348,155.392
C06965=1075.480,359.038,-99.461,175.544,30.354,155.393
C06966=1075.486,359.285,-99.496,175.548,30.359,155.394
C06967=1075.492,359.532,-99.533,175.551,30.365,155.395
C06968=1075.498,359.780,-99.570,175.555,30.371,155.397
C06969=1075.504,360.027,-99.606,175.558,30.377,155.398
C06970=1075.511,360.275,-99.643,175.562,30.383,155.399
C06971=1075.517,360.522,-99.680,175.565,30.389,155.400
C06972=1075.524,360.769,-99.716,175.569,30.395,155.401
C06973=1075.530,361.016,-99.752,175.573,30.401,155.402
C06974=1075.536,361.263,-99.789,175.576,30.407,155.403
C06975=1075.543,361.510,-99.825,175.580,30.413,155.404
C06976=1075.549,361.758,-99.863,175.583,30.419,155.406
C06977=1075.555,362.005,-99.899,175.587,30.425,155.407
C06978=1075.562,362.252,-99.936,175.590,30.431,155.408
C06979=1075.568,362.499,-99.972,175.595,30.437,155.409
C06980=1075.574,362.746,-100.009,175.598,30.442,155.410
C06981=1075.581,362.994,-100.045,175.602,30.448,155.411
C06982=1075.587,363.241,-100.083,175.605,30.454,155.412
C06983=1075.594,363.488,-100.120,175.609,30.460,155.414
C06984=1075.600,363.735,-100.156,175.612,30.466,155.415
C06985=1075.607,363.982,-100.193,175.617,30.472,155.416
C06986=1075.613,364.229,-100.230,175.620,30.478,155.417
C06987=1075.619,364.476,-100.267,175.624,30.484,155.418
C06988=1075.625,364.723,-100.303,175.627,30.491,155.420
C06989=1075.632,364.971,-100.340,175.630,30.497,155.421
C06990=1075.638,365.218,-100.378,175.635,30.503,155.422
C06991=1075.645,365.465,-100.414,175.638,30.509,155.423
C06992=1075.652,365.712,-100.452,175.642,30.515,155.424
C06993=1075.657,365.959,-100.489,175.645,30.521,155.425
C06994=1075.664,366.206,-100.525,175.649,30.527,155.427
C06995=1075.670,366.453,-100.563,175.653,30.534,155.428
C06996=1075.677,366.701,-100.600,175.657,30.540,155.429
C06997=1075.682,366.948,-100.638,175.660,30.546,155.430
C06998=1075.689,367.195,-100.674,175.664,30.552,155.432
C06999=1075.695,367.442,-100.712,175.668,30.559,155.433
C07000=1075.702,367.689,-100.749,175.672,30.565,155.434
C07001=1075.708,367.936,-100.786,175.675,30.571,155.435
C07002=1075.715,368.183,-100.824,175.679,30.578,155.436
C07003=1075.721,368.430,-100.861,175.682,30.584,155.438
C07004=1075.728,368.678,-100.899,175.687,30.590,155.439
C07005=1075.734,368.925,-100.935,175.690,30.596,155.440
C07006=1075.740,369.171,-100.973,175.693,30.603,155.441
C07007=1075.747,369.419,-101.010,175.698,30.609,155.442
C07008=1075.753,369.665,-101.048,175.701,30.615,155.444
C07009=1075.760,369.913,-101.085,175.705,30.622,155.445
C07010=1075.766,370.160,-101.123,175.708,30.628,155.446
C07011=1075.772,370.406,-101.160,175.713,30.634,155.448
C07012=1075.779,370.654,-101.198,175.716,30.641,155.449
C07013=1075.785,370.901,-101.235,175.720,30.647,155.450
C07014=1075.791,371.125,-101.269,175.723,30.653,155.451
C07015=1075.797,371.349,-101.304,175.727,30.659,155.452
C07016=1075.803,371.572,-101.337,175.730,30.665,155.453
C07017=1075.809,371.795,-101.372,175.734,30.671,155.455
C07018=1075.815,372.020,-101.405,175.737,30.676,155.456
C07019=1075.821,372.243,-101.440,175.741,30.682,155.457
C07020=1075.827,372.467,-101.473,175.745,30.688,155.458
C07021=1075.833,372.691,-101.508,175.747,30.694,155.459
C07022=1075.839,372.938,-101.546,175.752,30.700,155.460
C07023=1075.846,373.185,-101.583,175.755,30.707,155.462
C07024=1075.852,373.432,-101.621,175.759,30.713,155.463
C07025=1075.858,373.679,-101.659,175.763,30.720,155.464
C07026=1075.865,373.925,-101.696,175.767,30.726,155.466
C07027=1075.872,374.173,-101.735,175.770,30.733,155.467
C07028=1075.877,374.420,-101.772,175.774,30.740,155.468
C07029=1075.884,374.666,-101.811,175.778,30.746,155.470
C07030=1075.891,374.914,-101.849,175.781,30.753,155.471
C07031=1075.897,375.161,-101.887,175.786,30.760,155.472
C07032=1075.904,375.408,-101.925,175.789,30.766,155.474
C07033=1075.910,375.655,-101.962,175.794,30.773,155.475
C07034=1075.917,375.901,-102.001,175.797,30.780,155.476
C07035=1075.923,376.148,-102.039,175.801,30.786,155.478
C07036=1075.929,376.396,-102.077,175.805,30.793,155.479
C07037=1075.936,376.642,-102.116,175.809,30.800,155.480
C07038=1075.942,376.889,-102.154,175.812,30.806,155.482
C07039=1075.949,377.136,-102.192,175.817,30.814,155.483
C07040=1075.956,377.383,-102.230,175.820,30.820,155.484
C07041=1075.962,377.630,-102.268,175.825,30.827,155.486
C07042=1075.969,377.877,-102.307,175.828,30.834,155.487
C07043=1075.975,378.124,-102.345,175.832,30.840,155.488
C07044=1075.981,378.370,-102.383,175.836,30.848,155.490
C07045=1075.988,378.618,-102.421,175.840,30.855,155.491
C07046=1075.995,378.864,-102.460,175.844,30.861,155.493
C07047=1076.001,379.112,-102.498,175.848,30.868,155.494
C07048=1076.007,379.358,-102.537,175.852,30.875,155.495
C07049=1076.014,379.605,-102.576,175.856,30.882,155.497
C07050=1076.021,379.852,-102.614,175.859,30.889,155.498
C07051=1076.027,380.099,-102.652,175.864,30.896,155.500
C07052=1076.034,380.345,-102.690,175.867,30.903,155.501
C07053=1076.041,380.592,-102.728,175.872,30.910,155.502
C07054=1076.048,380.839,-102.767,175.875,30.917,155.504
C07055=1076.054,381.086,-102.806,175.880,30.924,155.505
C07056=1076.061,381.333,-102.845,175.883,30.931,155.507
C07057=1076.068,381.580,-102.883,175.888,30.938,155.508
C07058=1076.074,381.826,-102.922,175.891,30.945,155.509
C07059=1076.080,382.074,-102.961,175.896,30.952,155.511
C07060=1076.087,382.320,-103.000,175.899,30.959,155.512
C07061=1076.094,382.567,-103.039,175.904,30.966,155.514
C07062=1076.101,382.814,-103.078,175.907,30.973,155.515
C07063=1076.107,383.060,-103.116,175.912,30.980,155.517
C07064=1076.113,383.307,-103.155,175.915,30.987,155.518
C07065=1076.120,383.554,-103.194,175.920,30.995,155.520
C07066=1076.126,383.801,-103.233,175.923,31.002,155.521
C07067=1076.133,384.048,-103.272,175.928,31.009,155.523
C07068=1076.139,384.295,-103.311,175.931,31.016,155.524
C07069=1076.146,384.542,-103.350,175.936,31.024,155.526
C07070=1076.152,384.780,-103.388,175.939,31.031,155.527
C07071=1076.159,385.018,-103.426,175.943,31.038,155.528
C07072=1076.165,385.256,-103.463,175.947,31.045,155.530
C07073=1076.171,385.494,-103.501,175.951,31.052,155.531
C07074=1076.178,385.733,-103.539,175.954,31.059,155.533
C07075=1076.184,385.971,-103.577,175.959,31.066,155.534
C07076=1076.190,386.209,-103.614,175.963,31.073,155.536
C07077=1076.197,386.448,-103.653,175.967,31.080,155.537
C07078=1076.204,386.695,-103.691,175.971,31.088,155.539
C07079=1076.211,386.941,-103.731,175.975,31.095,155.540
C07080=1076.217,387.188,-103.770,175.979,31.103,155.542
C07081=1076.224,387.435,-103.809,175.983,31.110,155.543
C07082=1076.231,387.681,-103.849,175.988,31.117,155.545
C07083=1076.237,387.928,-103.888,175.991,31.125,155.546
C07084=1076.244,388.174,-103.928,175.996,31.132,155.548
C07085=1076.251,388.421,-103.967,175.999,31.140,155.549
C07086=1076.257,388.668,-104.006,176.004,31.147,155.551
C07087=1076.264,388.914,-104.046,176.008,31.155,155.552
C07088=1076.271,389.161,-104.086,176.012,31.162,155.554
C07089=1076.277,389.408,-104.125,176.016,31.170,155.556
C07090=1076.285,389.654,-104.164,176.020,31.178,155.557
C07091=1076.291,389.901,-104.204,176.024,31.185,155.559
C07092=1076.298,390.148,-104.243,176.029,31.193,155.560
C07093=1076.304,390.395,-104.283,176.033,31.200,155.562
C07094=1076.312,390.641,-104.322,176.037,31.208,155.563
C07095=1076.319,390.888,-104.362,176.042,31.216,155.565
C07096=1076.325,391.134,-104.402,176.045,31.223,155.567
C07097=1076.332,391.382,-104.441,176.050,31.231,155.568
C07098=1076.339,391.628,-104.482,176.054,31.239,155.570
C07099=1076.345,391.875,-104.522,176.058,31.247,155.571
C07100=1076.352,392.121,-104.561,176.062,31.255,155.573
C07101=1076.359,392.367,-104.601,176.067,31.262,155.575
C07102=1076.365,392.614,-104.640,176.070,31.270,155.576
C07103=1076.372,392.861,-104.681,176.075,31.278,155.578
C07104=1076.379,393.108,-104.721,176.079,31.286,155.580
C07105=1076.386,393.354,-104.760,176.084,31.294,155.581
C07106=1076.392,393.601,-104.801,176.088,31.302,155.583
C07107=1076.399,393.848,-104.841,176.092,31.310,155.585
C07108=1076.406,394.094,-104.881,176.097,31.318,155.586
C07109=1076.413,394.341,-104.921,176.100,31.325,155.588
C07110=1076.420,394.588,-104.961,176.105,31.334,155.590
C07111=1076.426,394.834,-105.001,176.109,31.342,155.591
C07112=1076.433,395.080,-105.041,176.114,31.350,155.593
C07113=1076.441,395.327,-105.082,176.117,31.357,155.595
C07114=1076.447,395.574,-105.122,176.122,31.366,155.596
C07115=1076.453,395.820,-105.163,176.127,31.374,155.598
C07116=1076.460,396.067,-105.203,176.130,31.382,155.600
C07117=1076.467,396.314,-105.243,176.135,31.390,155.601
C07118=1076.474,396.559,-105.283,176.139,31.398,155.603
C07119=1076.481,396.807,-105.324,176.144,31.406,155.605
C07120=1076.488,397.053,-105.364,176.148,31.415,155.607
C07121=1076.495,397.300,-105.405,176.152,31.423,155.608
C07122=1076.501,397.546,-105.445,176.157,31.431,155.610
C07123=1076.508,397.793,-105.486,176.161,31.439,155.612
C07124=1076.515,398.039,-105.527,176.166,31.448,155.614
C07125=1076.522,398.287,-105.567,176.169,31.456,155.615
C07126=1076.529,398.531,-105.607,176.174,31.464,155.617
C07127=1076.535,398.777,-105.648,176.178,31.473,155.619
C07128=1076.543,399.023,-105.688,176.183,31.481,155.621
C07129=1076.549,399.269,-105.729,176.188,31.489,155.622
C07130=1076.556,399.515,-105.770,176.191,31.498,155.624
C07131=1076.563,399.759,-105.810,176.196,31.506,155.626
C07132=1076.570,400.005,-105.851,176.200,31.515,155.628
C07133=1076.576,400.251,-105.892,176.205,31.523,155.630
C07134=1076.584,400.498,-105.933,176.210,31.532,155.631
C07135=1076.590,400.744,-105.973,176.214,31.540,155.633
C07136=1076.597,400.991,-106.014,176.218,31.549,155.635
C07137=1076.604,401.237,-106.055,176.222,31.557,155.637
C07138=1076.611,401.483,-106.096,176.227,31.566,155.639
C07139=1076.618,401.731,-106.137,176.232,31.574,155.641
C07140=1076.624,401.977,-106.178,176.236,31.583,155.643
C07141=1076.631,402.223,-106.220,176.241,31.592,155.644
C07142=1076.639,402.470,-106.261,176.245,31.601,155.646
C07143=1076.645,402.716,-106.302,176.250,31.609,155.648
C07144=1076.653,402.963,-106.343,176.255,31.618,155.650
C07145=1076.660,403.209,-106.384,176.259,31.627,155.652
C07146=1076.667,403.456,-106.425,176.263,31.636,155.654
C07147=1076.673,403.702,-106.467,176.267,31.644,155.656
C07148=1076.681,403.949,-106.508,176.272,31.653,155.658
C07149=1076.688,404.195,-106.549,176.277,31.662,155.659
C07150=1076.694,404.442,-106.591,176.281,31.671,155.661
C07151=1076.701,404.688,-106.632,176.286,31.680,155.663
C07152=1076.708,404.935,-106.673,176.290,31.689,155.665
C07153=1076.716,405.181,-106.714,176.295,31.698,155.667
C07154=1076.722,405.428,-106.756,176.300,31.707,155.669
C07155=1076.729,405.673,-106.798,176.304,31.716,155.671
C07156=1076.736,405.920,-106.840,176.309,31.725,155.673
C07157=1076.743,406.167,-106.881,176.314,31.734,155.675
C07158=1076.750,406.413,-106.922,176.318,31.743,155.677
C07159=1076.757,406.660,-106.965,176.323,31.752,155.679
C07160=1076.764,406.906,-107.006,176.328,31.761,155.681
C07161=1076.771,407.153,-107.048,176.332,31.771,155.683
C07162=1076.778,407.398,-107.089,176.337,31.780,155.685
C07163=1076.785,407.645,-107.131,176.341,31.789,155.687
C07164=1076.792,407.891,-107.173,176.346,31.798,155.689
C07165=1076.799,408.138,-107.215,176.352,31.808,155.691
C07166=1076.806,408.384,-107.257,176.356,31.817,155.693
C07167=1076.813,408.631,-107.299,176.361,31.826,155.695
C07168=1076.820,408.877,-107.341,176.366,31.836,155.697
C07169=1076.827,409.123,-107.383,176.370,31.845,155.699
C07170=1076.834,409.370,-107.425,176.375,31.855,155.701
C07171=1076.841,409.616,-107.467,176.380,31.864,155.703
C07172=1076.848,409.863,-107.510,176.384,31.874,155.705
C07173=1076.855,410.109,-107.551,176.389,31.883,155.707
C07174=1076.862,410.355,-107.593,176.394,31.892,155.710
C07175=1076.869,410.602,-107.636,176.399,31.902,155.712
C07176=1076.877,410.848,-107.678,176.404,31.911,155.714
C07177=1076.884,411.094,-107.720,176.409,31.921,155.716
C07178=1076.890,411.341,-107.762,176.414,31.931,155.718
C07179=1076.898,411.587,-107.804,176.418,31.940,155.720
C07180=1076.905,411.833,-107.847,176.424,31.950,155.722
C07181=1076.912,412.079,-107.889,176.429,31.960,155.724
C07182=1076.919,412.326,-107.932,176.433,31.970,155.726
C07183=1076.927,412.575,-107.975,176.438,31.979,155.729
C07184=1076.934,412.822,-108.017,176.443,31.989,155.731
C07185=1076.941,413.070,-108.060,176.448,31.999,155.733
C07186=1076.948,413.316,-108.102,176.453,32.009,155.735
C07187=1076.956,413.563,-108.145,176.458,32.019,155.737
C07188=1076.963,413.809,-108.188,176.464,32.029,155.740
C07189=1076.970,414.055,-108.230,176.468,32.039,155.742
C07190=1076.977,414.301,-108.272,176.473,32.049,155.744
C07191=1076.985,414.548,-108.316,176.478,32.058,155.746
C07192=1076.992,414.794,-108.358,176.483,32.068,155.748
C07193=1076.999,415.040,-108.400,176.488,32.078,155.750
C07194=1077.006,415.285,-108.444,176.493,32.088,155.753
C07195=1077.014,415.532,-108.486,176.499,32.099,155.755
C07196=1077.021,415.779,-108.529,176.503,32.109,155.757
C07197=1077.028,416.024,-108.572,176.508,32.119,155.760
C07198=1077.035,416.271,-108.615,176.514,32.129,155.762
C07199=1077.042,416.517,-108.658,176.519,32.139,155.764
C07200=1077.049,416.763,-108.701,176.523,32.150,155.766
C07201=1077.057,417.009,-108.744,176.529,32.160,155.769
C07202=1077.064,417.256,-108.787,176.534,32.170,155.771
C07203=1077.071,417.502,-108.830,176.540,32.181,155.773
C07204=1077.079,417.748,-108.874,176.544,32.191,155.776
C07205=1077.086,417.994,-108.917,176.549,32.201,155.778
C07206=1077.093,418.240,-108.960,176.555,32.212,155.780
C07207=1077.101,418.486,-109.003,176.560,32.222,155.783
C07208=1077.108,418.732,-109.047,176.566,32.233,155.785
C07209=1077.116,418.978,-109.090,176.570,32.243,155.787
C07210=1077.122,419.225,-109.133,176.576,32.254,155.790
C07211=1077.130,419.471,-109.176,176.581,32.265,155.792
C07212=1077.137,419.717,-109.220,176.587,32.275,155.794
C07213=1077.144,419.963,-109.264,176.592,32.286,155.797
C07214=1077.152,420.209,-109.307,176.597,32.297,155.799
C07215=1077.159,420.455,-109.351,176.602,32.307,155.802
C07216=1077.166,420.701,-109.394,176.608,32.318,155.804
C07217=1077.174,420.947,-109.438,176.613,32.329,155.807
C07218=1077.181,421.193,-109.481,176.619,32.340,155.809
C07219=1077.189,421.439,-109.525,176.623,32.350,155.811
C07220=1077.197,421.686,-109.568,176.629,32.361,155.814
C07221=1077.204,421.931,-109.613,176.634,32.372,155.816
C07222=1077.211,422.178,-109.656,176.640,32.383,155.819
C07223=1077.219,422.423,-109.700,176.645,32.394,155.821
C07224=1077.226,422.670,-109.744,176.651,32.405,155.824
C07225=1077.233,422.915,-109.788,176.656,32.416,155.826
C07226=1077.240,423.162,-109.832,176.661,32.428,155.829
C07227=1077.248,423.407,-109.876,176.667,32.439,155.831
C07228=1077.255,423.653,-109.920,176.673,32.450,155.834
C07229=1077.263,423.899,-109.965,176.678,32.461,155.837
C07230=1077.270,424.145,-110.008,176.684,32.472,155.839
C07231=1077.278,424.390,-110.052,176.689,32.484,155.842
C07232=1077.285,424.637,-110.096,176.695,32.495,155.844
C07233=1077.293,424.883,-110.141,176.700,32.506,155.847
C07234=1077.300,425.130,-110.185,176.706,32.518,155.849
C07235=1077.308,425.375,-110.229,176.711,32.529,155.852
C07236=1077.316,425.620,-110.273,176.717,32.540,155.855
C07237=1077.323,425.867,-110.317,176.723,32.552,155.857
C07238=1077.335,426.281,-110.393,176.732,32.571,155.862
C07239=1077.349,426.696,-110.468,176.742,32.591,155.866
C07240=1077.361,427.111,-110.542,176.752,32.611,155.871
C07241=1077.374,427.525,-110.617,176.762,32.630,155.875
C07242=1077.381,427.771,-110.662,176.767,32.642,155.878
C07243=1077.389,428.017,-110.707,176.773,32.654,155.881
C07244=1077.397,428.263,-110.752,176.779,32.666,155.883
C07245=1077.404,428.509,-110.797,176.784,32.677,155.886
C07246=1077.412,428.755,-110.841,176.790,32.690,155.889
C07247=1077.420,429.000,-110.887,176.795,32.701,155.892
C07248=1077.427,429.246,-110.931,176.801,32.713,155.894
C07249=1077.435,429.492,-110.976,176.807,32.726,155.897
C07250=1077.443,429.738,-111.021,176.813,32.738,155.900
C07251=1077.450,429.984,-111.066,176.819,32.750,155.903
C07252=1077.458,430.229,-111.111,176.825,32.762,155.906
C07253=1077.466,430.475,-111.156,176.831,32.774,155.908
C07254=1077.473,430.721,-111.201,176.837,32.786,155.911
C07255=1077.481,430.967,-111.246,176.844,32.799,155.914
C07256=1077.489,431.212,-111.291,176.850,32.811,155.917
C07257=1077.496,431.458,-111.336,176.856,32.823,155.920
C07258=1077.504,431.703,-111.382,176.862,32.836,155.923
C07259=1077.512,431.950,-111.427,176.868,32.848,155.926
C07260=1077.519,432.196,-111.473,176.874,32.860,155.928
C07261=1077.527,432.441,-111.518,176.880,32.873,155.931
